LIN {X 0,Y 116.665,Z 500.549,A -85,B 0,C 180,E1 -26190.852,E2 -26190.852} C_VEL
LIN {X 0,Y 112.984,Z 509.27,A -85,B 0,C 180,E1 -26195.582,E2 -26195.582} C_VEL
LIN {X 0,Y 109.778,Z 516.952,A -85,B 0,C 180,E1 -26201.06,E2 -26201.06} C_VEL
LIN {X 0,Y 107.278,Z 523.285,A -85,B 0,C 180,E1 -26207.132,E2 -26207.132} C_VEL
LIN {X 0,Y 105.67,Z 528.207,A -85,B 0,C 180,E1 -26213.504,E2 -26213.504} C_VEL
LIN {X 0,Y 104.773,Z 531.45,A -85,B 0,C 180,E1 -26219.305,E2 -26219.305} C_VEL
LIN {X 0,Y 105.042,Z 534.238,A -85,B 0,C 180,E1 -26227.006,E2 -26227.006} C_VEL
LIN {X 0,Y 106.467,Z 535.327,A -85,B 0,C 180,E1 -26233.438,E2 -26233.438} C_VEL
LIN {X 0,Y 109.318,Z 535.217,A -85,B 0,C 180,E1 -26240.463,E2 -26240.463} C_VEL
LIN {X 0,Y 112.597,Z 534.109,A -85,B 0,C 180,E1 -26245.822,E2 -26245.822} C_VEL
LIN {X 0,Y 117.145,Z 531.835,A -85,B 0,C 180,E1 -26251.317,E2 -26251.317} C_VEL
LIN {X 0,Y 122.747,Z 528.36,A -85,B 0,C 180,E1 -26256.372,E2 -26256.372} C_VEL
LIN {X 0,Y 129.145,Z 523.621,A -85,B 0,C 180,E1 -26260.942,E2 -26260.942} C_VEL
LIN {X 0,Y 136.15,Z 517.469,A -85,B 0,C 180,E1 -26265.043,E2 -26265.043} C_VEL
LIN {X 0,Y 143.911,Z 509.526,A -85,B 0,C 180,E1 -26268.735,E2 -26268.735} C_VEL
LIN {X 0,Y 150.719,Z 501.38,A -85,B 0,C 180,E1 -26271.527,E2 -26271.527} C_VEL
LIN {X 0,Y 157.259,Z 492.279,A -85,B 0,C 180,E1 -26273.801,E2 -26273.801} C_VEL
LIN {X 0,Y 163.793,Z 481.328,A -85,B 0,C 180,E1 -26275.864,E2 -26275.864} C_VEL
LIN {X 0,Y 169.141,Z 470.396,A -85,B 0,C 180,E1 -26277.418,E2 -26277.418} C_VEL
LIN {X 0,Y 173.622,Z 458.97,A -85,B 0,C 180,E1 -26278.608,E2 -26278.608} C_VEL
LIN {X 0,Y 177.377,Z 446.045,A -85,B 0,C 180,E1 -26279.628,E2 -26279.628} C_VEL
LIN {X 0,Y 180.062,Z 433.099,A -85,B 0,C 180,E1 -26280.239,E2 -26280.239} C_VEL
LIN {X 0,Y 181.656,Z 420.065,A -85,B 0,C 180,E1 -26280.703,E2 -26280.703} C_VEL
LIN {X 0,Y 179.793,Z 415.381,A -85,B 0,C 180,E1 -26283.473,E2 -26283.473} C_VEL
LIN {X 0,Y 178.027,Z 411.229,A -85,B 0,C 180,E1 -26286.802,E2 -26286.802} C_VEL
LIN {X 0,Y 177.28,Z 409.415,A -85,B 0,C 180,E1 -26288.729,E2 -26288.729} C_VEL
LIN {X 0,Y 176.009,Z 407.916,A -85,B 0,C 180,E1 -26293.862,E2 -26293.862} C_VEL
LIN {X 0,Y 175.948,Z 407.96,A -85,B 0,C 180,E1 -26297.086,E2 -26297.086} C_VEL
LIN {X 0,Y 176.976,Z 409.546,A -85,B 0,C 180,E1 -26302.087,E2 -26302.087} C_VEL
LIN {X 0,Y 178.38,Z 414.032,A -85,B 0,C 180,E1 -26305.887,E2 -26305.887} C_VEL
LIN {X 0,Y 179.645,Z 417.893,A -85,B 0,C 180,E1 -26308.255,E2 -26308.255} C_VEL
LIN {X 0,Y 181.323,Z 423.803,A -85,B 0,C 180,E1 -26310.965,E2 -26310.965} C_VEL
LIN {X 0,Y 178.937,Z 441.292,A -85,B 0,C 180,E1 -26311.578,E2 -26311.578} C_VEL
LIN {X 0,Y 175.823,Z 454.417,A -85,B 0,C 180,E1 -26312.249,E2 -26312.249} C_VEL
LIN {X 0,Y 171.93,Z 466.104,A -85,B 0,C 180,E1 -26313.093,E2 -26313.093} C_VEL
LIN {X 0,Y 166.888,Z 477.934,A -85,B 0,C 180,E1 -26314.284,E2 -26314.284} C_VEL
LIN {X 0,Y 161.219,Z 488.681,A -85,B 0,C 180,E1 -26315.736,E2 -26315.736} C_VEL
LIN {X 0,Y 155.145,Z 498.423,A -85,B 0,C 180,E1 -26317.576,E2 -26317.576} C_VEL
LIN {X 0,Y 148.601,Z 507.346,A -85,B 0,C 180,E1 -26319.796,E2 -26319.796} C_VEL
LIN {X 0,Y 142.303,Z 514.803,A -85,B 0,C 180,E1 -26322.217,E2 -26322.217} C_VEL
LIN {X 0,Y 135.314,Z 522.176,A -85,B 0,C 180,E1 -26325.497,E2 -26325.497} C_VEL
LIN {X 0,Y 128.731,Z 528.172,A -85,B 0,C 180,E1 -26329.087,E2 -26329.087} C_VEL
LIN {X 0,Y 122.68,Z 533.16,A -85,B 0,C 180,E1 -26333.323,E2 -26333.323} C_VEL
LIN {X 0,Y 117.749,Z 536.703,A -85,B 0,C 180,E1 -26337.524,E2 -26337.524} C_VEL
LIN {X 0,Y 112.044,Z 540.244,A -85,B 0,C 180,E1 -26343.97,E2 -26343.97} C_VEL
LIN {X 0,Y 107.971,Z 542.164,A -85,B 0,C 180,E1 -26351.021,E2 -26351.021} C_VEL
LIN {X 0,Y 105.791,Z 542.603,A -85,B 0,C 180,E1 -26358.518,E2 -26358.518} C_VEL
LIN {X 0,Y 105.297,Z 542.259,A -85,B 0,C 180,E1 -26362.342,E2 -26362.342} C_VEL
LIN {X 0,Y 105.199,Z 541.5,A -85,B 0,C 180,E1 -26366.182,E2 -26366.182} C_VEL
LIN {X 0,Y 105.382,Z 540.344,A -85,B 0,C 180,E1 -26370.012,E2 -26370.012} C_VEL
LIN {X 0,Y 105.287,Z 537.737,A -85,B 0,C 180,E1 -26375.759,E2 -26375.759} C_VEL
LIN {X 0,Y 105.847,Z 534.06,A -85,B 0,C 180,E1 -26381.502,E2 -26381.502} C_VEL
LIN {X 0,Y 107.216,Z 529.214,A -85,B 0,C 180,E1 -26387.168,E2 -26387.168} C_VEL
LIN {X 0,Y 109.582,Z 523.072,A -85,B 0,C 180,E1 -26392.643,E2 -26392.643} C_VEL
LIN {X 0,Y 112.775,Z 515.39,A -85,B 0,C 180,E1 -26397.876,E2 -26397.876} C_VEL
LIN {X 0,Y 115.509,Z 508.774,A -85,B 0,C 180,E1 -26401.396,E2 -26401.396} C_VEL
LIN {X 0,Y 119.502,Z 498.92,A -85,B 0,C 180,E1 -26405.514,E2 -26405.514} C_VEL
LIN {X 0,Y 123.418,Z 488.458,A -85,B 0,C 180,E1 -26408.795,E2 -26408.795} C_VEL
LIN {X 0,Y 127.343,Z 476.934,A -85,B 0,C 180,E1 -26411.484,E2 -26411.484} C_VEL
LIN {X 0,Y 129.324,Z 469.742,A -85,B 0,C 180,E1 -26412.819,E2 -26412.819} C_VEL
LIN {X 0,Y 130.256,Z 464.373,A -85,B 0,C 180,E1 -26413.78,E2 -26413.78} C_VEL
LIN {X 0,Y 129.985,Z 455.35,A -85,B 0,C 180,E1 -26415.619,E2 -26415.619} C_VEL
LIN {X 0,Y 129.24,Z 446.167,A -85,B 0,C 180,E1 -26417.279,E2 -26417.279} C_VEL
LIN {X 0,Y 129.425,Z 440.424,A -85,B 0,C 180,E1 -26417.922,E2 -26417.922} C_VEL
LIN {X 0,Y 132.785,Z 401.785,A -85,B 0,C 180,E1 -26419.9,E2 -26419.9} C_VEL
LIN {X 0,Y 132.575,Z 398.319,A -85,B 0,C 180,E1 -26420.249,E2 -26420.249} C_VEL
LIN {X 0,Y 127.688,Z 383.599,A -85,B 0,C 180,E1 -26423.302,E2 -26423.302} C_VEL
LIN {X 0,Y 122.637,Z 371.093,A -85,B 0,C 180,E1 -26426.647,E2 -26426.647} C_VEL
LIN {X 0,Y 118.748,Z 363.954,A -85,B 0,C 180,E1 -26429.275,E2 -26429.275} C_VEL
LIN {X 0,Y 113.441,Z 355.782,A -85,B 0,C 180,E1 -26433.186,E2 -26433.186} C_VEL
LIN {X 0,Y 111.169,Z 352.453,A -85,B 0,C 180,E1 -26435.068,E2 -26435.068} C_VEL
LIN {X 0,Y 108.638,Z 348.864,A -85,B 0,C 180,E1 -26437.286,E2 -26437.286} C_VEL
LIN {X 0,Y 105.705,Z 345.199,A -85,B 0,C 180,E1 -26440.078,E2 -26440.078} C_VEL
LIN {X 0,Y 104.68,Z 343.35,A -85,B 0,C 180,E1 -26441.226,E2 -26441.226} C_VEL
LIN {X 0,Y 102.272,Z 341.321,A -85,B 0,C 180,E1 -26443.808,E2 -26443.808} C_VEL
LIN {X 0,Y 101.161,Z 338.839,A -85,B 0,C 180,E1 -26445.351,E2 -26445.351} C_VEL
LIN {X 0,Y 100.982,Z 337.862,A -85,B 0,C 180,E1 -26445.818,E2 -26445.818} C_VEL
LIN {X 0,Y 101.24,Z 337.863,A -85,B 0,C 180,E1 -26452.019,E2 -26452.019} C_VEL
LIN {X 0,Y 101.844,Z 337.735,A -85,B 0,C 180,E1 -26460,E2 -26460} C_VEL
LIN {X 0,Y 101.234,Z 337.865,A -85,B 0,C 180,E1 -26467.981,E2 -26467.981} C_VEL
LIN {X 0,Y 101.064,Z 337.89,A -85,B 0,C 180,E1 -26473.164,E2 -26473.164} C_VEL
LIN {X 0,Y 100.778,Z 337.914,A -85,B 0,C 180,E1 -26480.407,E2 -26480.407} C_VEL
LIN {X 0,Y 100.715,Z 337.93,A -85,B 0,C 180,E1 -26484.863,E2 -26484.863} C_VEL
LIN {X 0,Y 100.651,Z 337.879,A -85,B 0,C 180,E1 -26493.063,E2 -26493.063} C_VEL
LIN {X 0,Y 100.637,Z 337.948,A -85,B 0,C 180,E1 -26499.793,E2 -26499.793} C_VEL
LIN {X 0,Y 100.608,Z 337.953,A -85,B 0,C 180,E1 -26506.537,E2 -26506.537} C_VEL
LIN {X 0,Y 101.477,Z 340.593,A -85,B 0,C 180,E1 -26507.943,E2 -26507.943} C_VEL
LIN {X 0,Y 103.656,Z 342.892,A -85,B 0,C 180,E1 -26510.43,E2 -26510.43} C_VEL
LIN {X 0,Y 104.88,Z 343.867,A -85,B 0,C 180,E1 -26511.687,E2 -26511.687} C_VEL
LIN {X 0,Y 106.673,Z 346.893,A -85,B 0,C 180,E1 -26513.621,E2 -26513.621} C_VEL
LIN {X 0,Y 108.718,Z 349.01,A -85,B 0,C 180,E1 -26515.473,E2 -26515.473} C_VEL
LIN {X 0,Y 111.229,Z 352.53,A -85,B 0,C 180,E1 -26517.66,E2 -26517.66} C_VEL
LIN {X 0,Y 115.759,Z 359.291,A -85,B 0,C 180,E1 -26521.274,E2 -26521.274} C_VEL
LIN {X 0,Y 119.958,Z 365.783,A -85,B 0,C 180,E1 -26524.211,E2 -26524.211} C_VEL
LIN {X 0,Y 126.98,Z 378.193,A -85,B 0,C 180,E1 -26528.608,E2 -26528.608} C_VEL
LIN {X 0,Y 133.38,Z 392.007,A -85,B 0,C 180,E1 -26532.218,E2 -26532.218} C_VEL
LIN {X 0,Y 129.761,Z 432.259,A -85,B 0,C 180,E1 -26534.216,E2 -26534.216} C_VEL
LIN {X 0,Y 127.732,Z 445.85,A -85,B 0,C 180,E1 -26535.452,E2 -26535.452} C_VEL
LIN {X 0,Y 124.976,Z 458.682,A -85,B 0,C 180,E1 -26537.197,E2 -26537.197} C_VEL
LIN {X 0,Y 121.513,Z 470.852,A -85,B 0,C 180,E1 -26539.497,E2 -26539.497} C_VEL
LIN {X 0,Y 117.767,Z 481.821,A -85,B 0,C 180,E1 -26542.273,E2 -26542.273} C_VEL
LIN {X 0,Y 113.927,Z 491.71,A -85,B 0,C 180,E1 -26545.566,E2 -26545.566} C_VEL
LIN {X 0,Y 109.663,Z 501.7,A -85,B 0,C 180,E1 -26549.988,E2 -26549.988} C_VEL
LIN {X 0,Y 105.832,Z 510.342,A -85,B 0,C 180,E1 -26555.052,E2 -26555.052} C_VEL
LIN {X 0,Y 102.535,Z 517.772,A -85,B 0,C 180,E1 -26560.851,E2 -26560.851} C_VEL
LIN {X 0,Y 100.35,Z 523.077,A -85,B 0,C 180,E1 -26566.254,E2 -26566.254} C_VEL
LIN {X 0,Y 98.774,Z 527.651,A -85,B 0,C 180,E1 -26572.333,E2 -26572.333} C_VEL
LIN {X 0,Y 97.814,Z 530.795,A -85,B 0,C 180,E1 -26577.824,E2 -26577.824} C_VEL
LIN {X 0,Y 97.714,Z 533.677,A -85,B 0,C 180,E1 -26585.108,E2 -26585.108} C_VEL
LIN {X 0,Y 98.401,Z 534.905,A -85,B 0,C 180,E1 -26589.98,E2 -26589.98} C_VEL
LIN {X 0,Y 99.836,Z 535.622,A -85,B 0,C 180,E1 -26595.254,E2 -26595.254} C_VEL
LIN {X 0,Y 102.768,Z 535.548,A -85,B 0,C 180,E1 -26602.013,E2 -26602.013} C_VEL
LIN {X 0,Y 107.044,Z 534.256,A -85,B 0,C 180,E1 -26608.566,E2 -26608.566} C_VEL
LIN {X 0,Y 111.831,Z 532.052,A -85,B 0,C 180,E1 -26613.902,E2 -26613.902} C_VEL
LIN {X 0,Y 117.929,Z 528.545,A -85,B 0,C 180,E1 -26619.049,E2 -26619.049} C_VEL
LIN {X 0,Y 124.838,Z 523.752,A -85,B 0,C 180,E1 -26623.651,E2 -26623.651} C_VEL
LIN {X 0,Y 132.368,Z 517.529,A -85,B 0,C 180,E1 -26627.738,E2 -26627.738} C_VEL
LIN {X 0,Y 140.548,Z 509.577,A -85,B 0,C 180,E1 -26631.372,E2 -26631.372} C_VEL
LIN {X 0,Y 148.293,Z 500.616,A -85,B 0,C 180,E1 -26634.283,E2 -26634.283} C_VEL
LIN {X 0,Y 154.89,Z 491.628,A -85,B 0,C 180,E1 -26636.388,E2 -26636.388} C_VEL
LIN {X 0,Y 161.675,Z 480.485,A -85,B 0,C 180,E1 -26638.372,E2 -26638.372} C_VEL
LIN {X 0,Y 167.387,Z 468.939,A -85,B 0,C 180,E1 -26639.869,E2 -26639.869} C_VEL
LIN {X 0,Y 172.181,Z 456.516,A -85,B 0,C 180,E1 -26641.067,E2 -26641.067} C_VEL
LIN {X 0,Y 175.631,Z 444.538,A -85,B 0,C 180,E1 -26641.915,E2 -26641.915} C_VEL
LIN {X 0,Y 178.261,Z 431.148,A -85,B 0,C 180,E1 -26642.472,E2 -26642.472} C_VEL
LIN {X 0,Y 179.109,Z 424.236,A -85,B 0,C 180,E1 -26642.752,E2 -26642.752} C_VEL
LIN {X 0,Y 177.663,Z 420.643,A -85,B 0,C 180,E1 -26645.224,E2 -26645.224} C_VEL
LIN {X 0,Y 176.617,Z 417.72,A -85,B 0,C 180,E1 -26647.664,E2 -26647.664} C_VEL
LIN {X 0,Y 176.084,Z 416.319,A -85,B 0,C 180,E1 -26649.187,E2 -26649.187} C_VEL
LIN {X 0,Y 175.003,Z 414.923,A -85,B 0,C 180,E1 -26653.943,E2 -26653.943} C_VEL
LIN {X 0,Y 174.957,Z 415.009,A -85,B 0,C 180,E1 -26657.186,E2 -26657.186} C_VEL
LIN {X 0,Y 175.803,Z 416.417,A -85,B 0,C 180,E1 -26661.627,E2 -26661.627} C_VEL
LIN {X 0,Y 177.023,Z 420.909,A -85,B 0,C 180,E1 -26665.342,E2 -26665.342} C_VEL
LIN {X 0,Y 178.184,Z 424.879,A -85,B 0,C 180,E1 -26667.725,E2 -26667.725} C_VEL
LIN {X 0,Y 178.797,Z 427.471,A -85,B 0,C 180,E1 -26668.905,E2 -26668.905} C_VEL
LIN {X 0,Y 176.708,Z 441.516,A -85,B 0,C 180,E1 -26669.408,E2 -26669.408} C_VEL
LIN {X 0,Y 173.682,Z 453.811,A -85,B 0,C 180,E1 -26670.006,E2 -26670.006} C_VEL
LIN {X 0,Y 169.713,Z 465.425,A -85,B 0,C 180,E1 -26670.786,E2 -26670.786} C_VEL
LIN {X 0,Y 164.502,Z 477.304,A -85,B 0,C 180,E1 -26671.906,E2 -26671.906} C_VEL
LIN {X 0,Y 157.966,Z 489.289,A -85,B 0,C 180,E1 -26673.488,E2 -26673.488} C_VEL
LIN {X 0,Y 150.979,Z 499.835,A -85,B 0,C 180,E1 -26675.471,E2 -26675.471} C_VEL
LIN {X 0,Y 144.214,Z 508.486,A -85,B 0,C 180,E1 -26677.656,E2 -26677.656} C_VEL
LIN {X 0,Y 137.676,Z 515.698,A -85,B 0,C 180,E1 -26680.049,E2 -26680.049} C_VEL
LIN {X 0,Y 130.37,Z 522.837,A -85,B 0,C 180,E1 -26683.32,E2 -26683.32} C_VEL
LIN {X 0,Y 123.463,Z 528.639,A -85,B 0,C 180,E1 -26686.933,E2 -26686.933} C_VEL
LIN {X 0,Y 116.658,Z 533.752,A -85,B 0,C 180,E1 -26691.552,E2 -26691.552} C_VEL
LIN {X 0,Y 111.833,Z 536.868,A -85,B 0,C 180,E1 -26695.574,E2 -26695.574} C_VEL
LIN {X 0,Y 108.521,Z 538.758,A -85,B 0,C 180,E1 -26698.812,E2 -26698.812} C_VEL
LIN {X 0,Y 103.228,Z 541.282,A -85,B 0,C 180,E1 -26705.905,E2 -26705.905} C_VEL
LIN {X 0,Y 99.829,Z 542.33,A -85,B 0,C 180,E1 -26713.659,E2 -26713.659} C_VEL
LIN {X 0,Y 98.838,Z 542.292,A -85,B 0,C 180,E1 -26717.698,E2 -26717.698} C_VEL
LIN {X 0,Y 98.111,Z 541.02,A -85,B 0,C 180,E1 -26725.906,E2 -26725.906} C_VEL
LIN {X 0,Y 98.305,Z 539.804,A -85,B 0,C 180,E1 -26730.013,E2 -26730.013} C_VEL
LIN {X 0,Y 98.221,Z 537.073,A -85,B 0,C 180,E1 -26736.174,E2 -26736.174} C_VEL
LIN {X 0,Y 98.884,Z 533.268,A -85,B 0,C 180,E1 -26742.324,E2 -26742.324} C_VEL
LIN {X 0,Y 100.421,Z 528.285,A -85,B 0,C 180,E1 -26748.369,E2 -26748.369} C_VEL
LIN {X 0,Y 103.044,Z 521.999,A -85,B 0,C 180,E1 -26754.168,E2 -26754.168} C_VEL
LIN {X 0,Y 106.495,Z 514.07,A -85,B 0,C 180,E1 -26759.678,E2 -26759.678} C_VEL
LIN {X 0,Y 110.42,Z 505.227,A -85,B 0,C 180,E1 -26764.308,E2 -26764.308} C_VEL
LIN {X 0,Y 114.237,Z 496.074,A -85,B 0,C 180,E1 -26767.979,E2 -26767.979} C_VEL
LIN {X 0,Y 118.457,Z 485.04,A -85,B 0,C 180,E1 -26771.314,E2 -26771.314} C_VEL
LIN {X 0,Y 122.03,Z 474.28,A -85,B 0,C 180,E1 -26773.729,E2 -26773.729} C_VEL
LIN {X 0,Y 125.551,Z 461.419,A -85,B 0,C 180,E1 -26775.836,E2 -26775.836} C_VEL
LIN {X 0,Y 128.155,Z 448.849,A -85,B 0,C 180,E1 -26777.257,E2 -26777.257} C_VEL
LIN {X 0,Y 129.425,Z 440.424,A -85,B 0,C 180,E1 -26777.922,E2 -26777.922} C_VEL
LIN {X 0,Y 129.569,Z 434.661,A -85,B 0,C 180,E1 -26778.478,E2 -26778.478} C_VEL
LIN {X 0,Y 126.8,Z 415.841,A -85,B 0,C 180,E1 -26780.976,E2 -26780.976} C_VEL
LIN {X 0,Y 126.704,Z 410.024,A -85,B 0,C 180,E1 -26781.472,E2 -26781.472} C_VEL
LIN {X 0,Y 127.263,Z 400.819,A -85,B 0,C 180,E1 -26782.022,E2 -26782.022} C_VEL
LIN {X 0,Y 122.632,Z 386.514,A -85,B 0,C 180,E1 -26785.221,E2 -26785.221} C_VEL
LIN {X 0,Y 117.719,Z 374.148,A -85,B 0,C 180,E1 -26788.789,E2 -26788.789} C_VEL
LIN {X 0,Y 112.832,Z 365.521,A -85,B 0,C 180,E1 -26792.465,E2 -26792.465} C_VEL
LIN {X 0,Y 108.275,Z 358.439,A -85,B 0,C 180,E1 -26796.346,E2 -26796.346} C_VEL
LIN {X 0,Y 104.809,Z 353.675,A -85,B 0,C 180,E1 -26799.643,E2 -26799.643} C_VEL
LIN {X 0,Y 102.41,Z 350.065,A -85,B 0,C 180,E1 -26802.299,E2 -26802.299} C_VEL
LIN {X 0,Y 99.45,Z 346.857,A -85,B 0,C 180,E1 -26805.81,E2 -26805.81} C_VEL
LIN {X 0,Y 98.251,Z 344.352,A -85,B 0,C 180,E1 -26807.608,E2 -26807.608} C_VEL
LIN {X 0,Y 95.865,Z 342.587,A -85,B 0,C 180,E1 -26811.038,E2 -26811.038} C_VEL
LIN {X 0,Y 94.427,Z 339.863,A -85,B 0,C 180,E1 -26813.858,E2 -26813.858} C_VEL
LIN {X 0,Y 94.233,Z 338.69,A -85,B 0,C 180,E1 -26814.651,E2 -26814.651} C_VEL
LIN {X 0,Y 94.773,Z 338.613,A -85,B 0,C 180,E1 -26820,E2 -26820} C_VEL
LIN {X 0,Y 94.145,Z 338.742,A -85,B 0,C 180,E1 -26828.587,E2 -26828.587} C_VEL
LIN {X 0,Y 93.972,Z 338.775,A -85,B 0,C 180,E1 -26833.487,E2 -26833.487} C_VEL
LIN {X 0,Y 93.645,Z 338.814,A -85,B 0,C 180,E1 -26842.04,E2 -26842.04} C_VEL
LIN {X 0,Y 93.555,Z 338.791,A -85,B 0,C 180,E1 -26846.791,E2 -26846.791} C_VEL
LIN {X 0,Y 93.556,Z 338.77,A -85,B 0,C 180,E1 -26854.257,E2 -26854.257} C_VEL
LIN {X 0,Y 93.533,Z 338.972,A -85,B 0,C 180,E1 -26857.071,E2 -26857.071} C_VEL
LIN {X 0,Y 94.242,Z 341.088,A -85,B 0,C 180,E1 -26858.806,E2 -26858.806} C_VEL
LIN {X 0,Y 96.082,Z 343.431,A -85,B 0,C 180,E1 -26862.095,E2 -26862.095} C_VEL
LIN {X 0,Y 98.178,Z 344.839,A -85,B 0,C 180,E1 -26865.067,E2 -26865.067} C_VEL
LIN {X 0,Y 99.749,Z 347.721,A -85,B 0,C 180,E1 -26867.341,E2 -26867.341} C_VEL
LIN {X 0,Y 102.304,Z 350.218,A -85,B 0,C 180,E1 -26870.284,E2 -26870.284} C_VEL
LIN {X 0,Y 104.479,Z 353.509,A -85,B 0,C 180,E1 -26872.729,E2 -26872.729} C_VEL
LIN {X 0,Y 106.069,Z 355.432,A -85,B 0,C 180,E1 -26874.296,E2 -26874.296} C_VEL
LIN {X 0,Y 109.432,Z 360.383,A -85,B 0,C 180,E1 -26877.391,E2 -26877.391} C_VEL
LIN {X 0,Y 113.983,Z 367.303,A -85,B 0,C 180,E1 -26881.098,E2 -26881.098} C_VEL
LIN {X 0,Y 120.248,Z 378.29,A -85,B 0,C 180,E1 -26885.559,E2 -26885.559} C_VEL
LIN {X 0,Y 124.203,Z 386.015,A -85,B 0,C 180,E1 -26888.1,E2 -26888.1} C_VEL
LIN {X 0,Y 127.722,Z 394.162,A -85,B 0,C 180,E1 -26890.271,E2 -26890.271} C_VEL
LIN {X 0,Y 124.17,Z 432.589,A -85,B 0,C 180,E1 -26892.243,E2 -26892.243} C_VEL
LIN {X 0,Y 122.087,Z 445.935,A -85,B 0,C 180,E1 -26893.477,E2 -26893.477} C_VEL
LIN {X 0,Y 119.216,Z 458.812,A -85,B 0,C 180,E1 -26895.262,E2 -26895.262} C_VEL
LIN {X 0,Y 115.342,Z 471.772,A -85,B 0,C 180,E1 -26897.791,E2 -26897.791} C_VEL
LIN {X 0,Y 111.105,Z 483.373,A -85,B 0,C 180,E1 -26900.89,E2 -26900.89} C_VEL
LIN {X 0,Y 106.412,Z 494.631,A -85,B 0,C 180,E1 -26905.03,E2 -26905.03} C_VEL
LIN {X 0,Y 101.85,Z 504.567,A -85,B 0,C 180,E1 -26909.987,E2 -26909.987} C_VEL
LIN {X 0,Y 98.237,Z 512.27,A -85,B 0,C 180,E1 -26915.14,E2 -26915.14} C_VEL
LIN {X 0,Y 94.783,Z 519.726,A -85,B 0,C 180,E1 -26921.751,E2 -26921.751} C_VEL
LIN {X 0,Y 92.75,Z 524.709,A -85,B 0,C 180,E1 -26927.628,E2 -26927.628} C_VEL
LIN {X 0,Y 91.123,Z 529.462,A -85,B 0,C 180,E1 -26935.08,E2 -26935.08} C_VEL
LIN {X 0,Y 90.508,Z 532.89,A -85,B 0,C 180,E1 -26942.906,E2 -26942.906} C_VEL
LIN {X 0,Y 91.201,Z 534.814,A -85,B 0,C 180,E1 -26949.592,E2 -26949.592} C_VEL
LIN {X 0,Y 93.339,Z 535.914,A -85,B 0,C 180,E1 -26957.339,E2 -26957.339} C_VEL
LIN {X 0,Y 96.695,Z 535.815,A -85,B 0,C 180,E1 -26964.447,E2 -26964.447} C_VEL
LIN {X 0,Y 101.187,Z 534.601,A -85,B 0,C 180,E1 -26970.909,E2 -26970.909} C_VEL
LIN {X 0,Y 106.958,Z 532.196,A -85,B 0,C 180,E1 -26976.872,E2 -26976.872} C_VEL
LIN {X 0,Y 113.405,Z 528.751,A -85,B 0,C 180,E1 -26981.949,E2 -26981.949} C_VEL
LIN {X 0,Y 120.858,Z 523.923,A -85,B 0,C 180,E1 -26986.549,E2 -26986.549} C_VEL
LIN {X 0,Y 128.934,Z 517.602,A -85,B 0,C 180,E1 -26990.588,E2 -26990.588} C_VEL
LIN {X 0,Y 137.509,Z 509.619,A -85,B 0,C 180,E1 -26994.133,E2 -26994.133} C_VEL
LIN {X 0,Y 145.148,Z 501.198,A -85,B 0,C 180,E1 -26996.768,E2 -26996.768} C_VEL
LIN {X 0,Y 152.847,Z 491.087,A -85,B 0,C 180,E1 -26999.034,E2 -26999.034} C_VEL
LIN {X 0,Y 159.337,Z 480.758,A -85,B 0,C 180,E1 -27000.789,E2 -27000.789} C_VEL
LIN {X 0,Y 165.215,Z 469.244,A -85,B 0,C 180,E1 -27002.211,E2 -27002.211} C_VEL
LIN {X 0,Y 170.202,Z 456.677,A -85,B 0,C 180,E1 -27003.368,E2 -27003.368} C_VEL
LIN {X 0,Y 173.868,Z 444.229,A -85,B 0,C 180,E1 -27004.187,E2 -27004.187} C_VEL
LIN {X 0,Y 176.467,Z 431.106,A -85,B 0,C 180,E1 -27004.685,E2 -27004.685} C_VEL
LIN {X 0,Y 176.792,Z 428.711,A -85,B 0,C 180,E1 -27004.793,E2 -27004.793} C_VEL
LIN {X 0,Y 175.338,Z 424.442,A -85,B 0,C 180,E1 -27008.282,E2 -27008.282} C_VEL
LIN {X 0,Y 174.758,Z 423.035,A -85,B 0,C 180,E1 -27010.067,E2 -27010.067} C_VEL
LIN {X 0,Y 173.975,Z 421.931,A -85,B 0,C 180,E1 -27014.229,E2 -27014.229} C_VEL
LIN {X 0,Y 173.963,Z 422.087,A -85,B 0,C 180,E1 -27017.287,E2 -27017.287} C_VEL
LIN {X 0,Y 174.653,Z 423.395,A -85,B 0,C 180,E1 -27021.233,E2 -27021.233} C_VEL
LIN {X 0,Y 175.67,Z 427.597,A -85,B 0,C 180,E1 -27024.681,E2 -27024.681} C_VEL
LIN {X 0,Y 176.53,Z 431.263,A -85,B 0,C 180,E1 -27026.802,E2 -27026.802} C_VEL
LIN {X 0,Y 174.269,Z 443.994,A -85,B 0,C 180,E1 -27027.26,E2 -27027.26} C_VEL
LIN {X 0,Y 170.647,Z 457.145,A -85,B 0,C 180,E1 -27027.93,E2 -27027.93} C_VEL
LIN {X 0,Y 166.284,Z 468.708,A -85,B 0,C 180,E1 -27028.741,E2 -27028.741} C_VEL
LIN {X 0,Y 160.965,Z 479.778,A -85,B 0,C 180,E1 -27029.822,E2 -27029.822} C_VEL
LIN {X 0,Y 154.23,Z 491.13,A -85,B 0,C 180,E1 -27031.329,E2 -27031.329} C_VEL
LIN {X 0,Y 147.028,Z 501.279,A -85,B 0,C 180,E1 -27033.249,E2 -27033.249} C_VEL
LIN {X 0,Y 138.691,Z 511.07,A -85,B 0,C 180,E1 -27035.85,E2 -27035.85} C_VEL
LIN {X 0,Y 133.26,Z 516.604,A -85,B 0,C 180,E1 -27037.734,E2 -27037.734} C_VEL
LIN {X 0,Y 125.632,Z 523.503,A -85,B 0,C 180,E1 -27040.977,E2 -27040.977} C_VEL
LIN {X 0,Y 118.392,Z 529.106,A -85,B 0,C 180,E1 -27044.594,E2 -27044.594} C_VEL
LIN {X 0,Y 110.781,Z 534.254,A -85,B 0,C 180,E1 -27049.578,E2 -27049.578} C_VEL
LIN {X 0,Y 106.043,Z 537.026,A -85,B 0,C 180,E1 -27053.4,E2 -27053.4} C_VEL
LIN {X 0,Y 102.504,Z 538.794,A -85,B 0,C 180,E1 -27056.753,E2 -27056.753} C_VEL
LIN {X 0,Y 96.784,Z 541.179,A -85,B 0,C 180,E1 -27064.188,E2 -27064.188} C_VEL
LIN {X 0,Y 94.585,Z 541.817,A -85,B 0,C 180,E1 -27068.207,E2 -27068.207} C_VEL
LIN {X 0,Y 91.882,Z 541.932,A -85,B 0,C 180,E1 -27076.75,E2 -27076.75} C_VEL
LIN {X 0,Y 91.04,Z 540.541,A -85,B 0,C 180,E1 -27085.587,E2 -27085.587} C_VEL
LIN {X 0,Y 91.215,Z 539.262,A -85,B 0,C 180,E1 -27090.014,E2 -27090.014} C_VEL
LIN {X 0,Y 91.178,Z 536.404,A -85,B 0,C 180,E1 -27096.653,E2 -27096.653} C_VEL
LIN {X 0,Y 91.953,Z 532.461,A -85,B 0,C 180,E1 -27103.269,E2 -27103.269} C_VEL
LIN {X 0,Y 94.061,Z 526.314,A -85,B 0,C 180,E1 -27110.801,E2 -27110.801} C_VEL
LIN {X 0,Y 97.096,Z 519.568,A -85,B 0,C 180,E1 -27116.91,E2 -27116.91} C_VEL
LIN {X 0,Y 101.007,Z 511.143,A -85,B 0,C 180,E1 -27122.645,E2 -27122.645} C_VEL
LIN {X 0,Y 105.05,Z 502.467,A -85,B 0,C 180,E1 -27127.034,E2 -27127.034} C_VEL
LIN {X 0,Y 109.683,Z 491.788,A -85,B 0,C 180,E1 -27131.067,E2 -27131.067} C_VEL
LIN {X 0,Y 113.774,Z 481.222,A -85,B 0,C 180,E1 -27134.034,E2 -27134.034} C_VEL
LIN {X 0,Y 117.534,Z 469.483,A -85,B 0,C 180,E1 -27136.482,E2 -27136.482} C_VEL
LIN {X 0,Y 121.012,Z 456.231,A -85,B 0,C 180,E1 -27138.407,E2 -27138.407} C_VEL
LIN {X 0,Y 123.437,Z 442.968,A -85,B 0,C 180,E1 -27139.716,E2 -27139.716} C_VEL
LIN {X 0,Y 124.987,Z 428.585,A -85,B 0,C 180,E1 -27140.583,E2 -27140.583} C_VEL
LIN {X 0,Y 126.704,Z 410.024,A -85,B 0,C 180,E1 -27141.472,E2 -27141.472} C_VEL
LIN {X 0,Y 126.409,Z 406.934,A -85,B 0,C 180,E1 -27141.844,E2 -27141.844} C_VEL
LIN {X 0,Y 124.852,Z 403.138,A -85,B 0,C 180,E1 -27142.79,E2 -27142.79} C_VEL
LIN {X 0,Y 119.609,Z 394.847,A -85,B 0,C 180,E1 -27145.852,E2 -27145.852} C_VEL
LIN {X 0,Y 118.966,Z 393.121,A -85,B 0,C 180,E1 -27146.326,E2 -27146.326} C_VEL
LIN {X 0,Y 114.902,Z 381.895,A -85,B 0,C 180,E1 -27149.496,E2 -27149.496} C_VEL
LIN {X 0,Y 112.445,Z 376.399,A -85,B 0,C 180,E1 -27151.486,E2 -27151.486} C_VEL
LIN {X 0,Y 107.195,Z 367.318,A -85,B 0,C 180,E1 -27156,E2 -27156} C_VEL
LIN {X 0,Y 104.558,Z 363.42,A -85,B 0,C 180,E1 -27158.499,E2 -27158.499} C_VEL
LIN {X 0,Y 101.95,Z 359.506,A -85,B 0,C 180,E1 -27161.288,E2 -27161.288} C_VEL
LIN {X 0,Y 99.407,Z 355.75,A -85,B 0,C 180,E1 -27164.363,E2 -27164.363} C_VEL
LIN {X 0,Y 97,Z 352.843,A -85,B 0,C 180,E1 -27167.517,E2 -27167.517} C_VEL
LIN {X 0,Y 95.944,Z 350.818,A -85,B 0,C 180,E1 -27169.221,E2 -27169.221} C_VEL
LIN {X 0,Y 93.656,Z 348.585,A -85,B 0,C 180,E1 -27172.996,E2 -27172.996} C_VEL
LIN {X 0,Y 92.25,Z 345.466,A -85,B 0,C 180,E1 -27176.178,E2 -27176.178} C_VEL
LIN {X 0,Y 89.759,Z 343.985,A -85,B 0,C 180,E1 -27182.244,E2 -27182.244} C_VEL
LIN {X 0,Y 87.815,Z 342.206,A -85,B 0,C 180,E1 -27191.542,E2 -27191.542} C_VEL
LIN {X 0,Y 87.56,Z 342.303,A -85,B 0,C 180,E1 -27197.519,E2 -27197.519} C_VEL
LIN {X 0,Y 88.537,Z 343.801,A -85,B 0,C 180,E1 -27206.273,E2 -27206.273} C_VEL
LIN {X 0,Y 91.71,Z 345.783,A -85,B 0,C 180,E1 -27215.572,E2 -27215.572} C_VEL
LIN {X 0,Y 93.334,Z 349.009,A -85,B 0,C 180,E1 -27219.256,E2 -27219.256} C_VEL
LIN {X 0,Y 96.005,Z 351.432,A -85,B 0,C 180,E1 -27223.653,E2 -27223.653} C_VEL
LIN {X 0,Y 98.151,Z 354.799,A -85,B 0,C 180,E1 -27226.842,E2 -27226.842} C_VEL
LIN {X 0,Y 99.878,Z 356.67,A -85,B 0,C 180,E1 -27228.959,E2 -27228.959} C_VEL
LIN {X 0,Y 102.316,Z 360.108,A -85,B 0,C 180,E1 -27231.802,E2 -27231.802} C_VEL
LIN {X 0,Y 106.016,Z 365.626,A -85,B 0,C 180,E1 -27235.605,E2 -27235.605} C_VEL
LIN {X 0,Y 110.606,Z 372.915,A -85,B 0,C 180,E1 -27239.647,E2 -27239.647} C_VEL
LIN {X 0,Y 116.454,Z 383.683,A -85,B 0,C 180,E1 -27244.187,E2 -27244.187} C_VEL
LIN {X 0,Y 120.174,Z 391.293,A -85,B 0,C 180,E1 -27246.748,E2 -27246.748} C_VEL
LIN {X 0,Y 122.315,Z 396.762,A -85,B 0,C 180,E1 -27248.232,E2 -27248.232} C_VEL
LIN {X 0,Y 118.78,Z 432.764,A -85,B 0,C 180,E1 -27250.083,E2 -27250.083} C_VEL
LIN {X 0,Y 116.533,Z 446.408,A -85,B 0,C 180,E1 -27251.361,E2 -27251.361} C_VEL
LIN {X 0,Y 113.599,Z 458.946,A -85,B 0,C 180,E1 -27253.131,E2 -27253.131} C_VEL
LIN {X 0,Y 109.652,Z 471.598,A -85,B 0,C 180,E1 -27255.639,E2 -27255.639} C_VEL
LIN {X 0,Y 105.081,Z 483.561,A -85,B 0,C 180,E1 -27258.902,E2 -27258.902} C_VEL
LIN {X 0,Y 100.583,Z 493.822,A -85,B 0,C 180,E1 -27262.754,E2 -27262.754} C_VEL
LIN {X 0,Y 95.745,Z 503.922,A -85,B 0,C 180,E1 -27267.883,E2 -27267.883} C_VEL
LIN {X 0,Y 91.555,Z 512.273,A -85,B 0,C 180,E1 -27273.694,E2 -27273.694} C_VEL
LIN {X 0,Y 88.109,Z 519.258,A -85,B 0,C 180,E1 -27280.212,E2 -27280.212} C_VEL
LIN {X 0,Y 85.818,Z 524.466,A -85,B 0,C 180,E1 -27286.639,E2 -27286.639} C_VEL
LIN {X 0,Y 84.045,Z 529.341,A -85,B 0,C 180,E1 -27294.696,E2 -27294.696} C_VEL
LIN {X 0,Y 83.416,Z 532.717,A -85,B 0,C 180,E1 -27302.592,E2 -27302.592} C_VEL
LIN {X 0,Y 84.472,Z 535.184,A -85,B 0,C 180,E1 -27311.704,E2 -27311.704} C_VEL
LIN {X 0,Y 86.969,Z 536.207,A -85,B 0,C 180,E1 -27319.723,E2 -27319.723} C_VEL
LIN {X 0,Y 91.247,Z 536.02,A -85,B 0,C 180,E1 -27327.879,E2 -27327.879} C_VEL
LIN {X 0,Y 95.877,Z 534.854,A -85,B 0,C 180,E1 -27333.908,E2 -27333.908} C_VEL
LIN {X 0,Y 102.089,Z 532.498,A -85,B 0,C 180,E1 -27339.866,E2 -27339.866} C_VEL
LIN {X 0,Y 109.246,Z 528.957,A -85,B 0,C 180,E1 -27345.088,E2 -27345.088} C_VEL
LIN {X 0,Y 117.208,Z 524.089,A -85,B 0,C 180,E1 -27349.637,E2 -27349.637} C_VEL
LIN {X 0,Y 125.819,Z 517.714,A -85,B 0,C 180,E1 -27353.586,E2 -27353.586} C_VEL
LIN {X 0,Y 134.887,Z 509.682,A -85,B 0,C 180,E1 -27357.013,E2 -27357.013} C_VEL
LIN {X 0,Y 143.164,Z 500.83,A -85,B 0,C 180,E1 -27359.623,E2 -27359.623} C_VEL
LIN {X 0,Y 151.138,Z 490.617,A -85,B 0,C 180,E1 -27361.738,E2 -27361.738} C_VEL
LIN {X 0,Y 157.479,Z 480.741,A -85,B 0,C 180,E1 -27363.301,E2 -27363.301} C_VEL
LIN {X 0,Y 163.758,Z 468.629,A -85,B 0,C 180,E1 -27364.701,E2 -27364.701} C_VEL
LIN {X 0,Y 168.983,Z 455.651,A -85,B 0,C 180,E1 -27365.802,E2 -27365.802} C_VEL
LIN {X 0,Y 172.463,Z 443.822,A -85,B 0,C 180,E1 -27366.507,E2 -27366.507} C_VEL
LIN {X 0,Y 174.623,Z 433.497,A -85,B 0,C 180,E1 -27366.935,E2 -27366.935} C_VEL
LIN {X 0,Y 174.034,Z 431.179,A -85,B 0,C 180,E1 -27368.879,E2 -27368.879} C_VEL
LIN {X 0,Y 173.616,Z 429.961,A -85,B 0,C 180,E1 -27370.406,E2 -27370.406} C_VEL
LIN {X 0,Y 172.991,Z 428.952,A -85,B 0,C 180,E1 -27374.108,E2 -27374.108} C_VEL
LIN {X 0,Y 173.008,Z 429.226,A -85,B 0,C 180,E1 -27377.779,E2 -27377.779} C_VEL
LIN {X 0,Y 173.454,Z 430.197,A -85,B 0,C 180,E1 -27380.599,E2 -27380.599} C_VEL
LIN {X 0,Y 174.238,Z 434.193,A -85,B 0,C 180,E1 -27383.946,E2 -27383.946} C_VEL
LIN {X 0,Y 174.407,Z 435.684,A -85,B 0,C 180,E1 -27384.714,E2 -27384.714} C_VEL
LIN {X 0,Y 171.458,Z 448.876,A -85,B 0,C 180,E1 -27385.184,E2 -27385.184} C_VEL
LIN {X 0,Y 167.023,Z 462.397,A -85,B 0,C 180,E1 -27385.914,E2 -27385.914} C_VEL
LIN {X 0,Y 161.478,Z 474.901,A -85,B 0,C 180,E1 -27386.872,E2 -27386.872} C_VEL
LIN {X 0,Y 154.522,Z 487.26,A -85,B 0,C 180,E1 -27388.236,E2 -27388.236} C_VEL
LIN {X 0,Y 147.74,Z 497.119,A -85,B 0,C 180,E1 -27389.78,E2 -27389.78} C_VEL
LIN {X 0,Y 140.406,Z 506.087,A -85,B 0,C 180,E1 -27391.711,E2 -27391.711} C_VEL
LIN {X 0,Y 131.827,Z 514.909,A -85,B 0,C 180,E1 -27394.299,E2 -27394.299} C_VEL
LIN {X 0,Y 123.763,Z 522.052,A -85,B 0,C 180,E1 -27397.367,E2 -27397.367} C_VEL
LIN {X 0,Y 116.004,Z 527.885,A -85,B 0,C 180,E1 -27400.795,E2 -27400.795} C_VEL
LIN {X 0,Y 108.866,Z 532.543,A -85,B 0,C 180,E1 -27404.776,E2 -27404.776} C_VEL
LIN {X 0,Y 103.296,Z 535.699,A -85,B 0,C 180,E1 -27408.655,E2 -27408.655} C_VEL
LIN {X 0,Y 96.637,Z 538.838,A -85,B 0,C 180,E1 -27414.442,E2 -27414.442} C_VEL
LIN {X 0,Y 90.416,Z 541.074,A -85,B 0,C 180,E1 -27422.219,E2 -27422.219} C_VEL
LIN {X 0,Y 86.232,Z 541.769,A -85,B 0,C 180,E1 -27430.991,E2 -27430.991} C_VEL
LIN {X 0,Y 84.226,Z 540.995,A -85,B 0,C 180,E1 -27440.41,E2 -27440.41} C_VEL
LIN {X 0,Y 83.965,Z 540.046,A -85,B 0,C 180,E1 -27445.215,E2 -27445.215} C_VEL
LIN {X 0,Y 84.132,Z 538.661,A -85,B 0,C 180,E1 -27450.016,E2 -27450.016} C_VEL
LIN {X 0,Y 84.115,Z 535.69,A -85,B 0,C 180,E1 -27457.215,E2 -27457.215} C_VEL
LIN {X 0,Y 85.02,Z 531.609,A -85,B 0,C 180,E1 -27464.373,E2 -27464.373} C_VEL
LIN {X 0,Y 87.438,Z 525.281,A -85,B 0,C 180,E1 -27472.459,E2 -27472.459} C_VEL
LIN {X 0,Y 90.783,Z 518.36,A -85,B 0,C 180,E1 -27478.951,E2 -27478.951} C_VEL
LIN {X 0,Y 94.3,Z 511.258,A -85,B 0,C 180,E1 -27483.998,E2 -27483.998} C_VEL
LIN {X 0,Y 98.439,Z 502.879,A -85,B 0,C 180,E1 -27488.542,E2 -27488.542} C_VEL
LIN {X 0,Y 103.386,Z 492.103,A -85,B 0,C 180,E1 -27492.84,E2 -27492.84} C_VEL
LIN {X 0,Y 107.632,Z 481.644,A -85,B 0,C 180,E1 -27495.925,E2 -27495.925} C_VEL
LIN {X 0,Y 111.584,Z 470.18,A -85,B 0,C 180,E1 -27498.425,E2 -27498.425} C_VEL
LIN {X 0,Y 114.855,Z 458.44,A -85,B 0,C 180,E1 -27500.251,E2 -27500.251} C_VEL
LIN {X 0,Y 117.642,Z 445.095,A -85,B 0,C 180,E1 -27501.673,E2 -27501.673} C_VEL
LIN {X 0,Y 119.274,Z 432.314,A -85,B 0,C 180,E1 -27502.547,E2 -27502.547} C_VEL
LIN {X 0,Y 121.913,Z 402.898,A -85,B 0,C 180,E1 -27504.054,E2 -27504.054} C_VEL
LIN {X 0,Y 118.966,Z 393.121,A -85,B 0,C 180,E1 -27506.326,E2 -27506.326} C_VEL
LIN {X 0,Y 117.678,Z 389.959,A -85,B 0,C 180,E1 -27507.266,E2 -27507.266} C_VEL
LIN {X 0,Y 115.053,Z 386.01,A -85,B 0,C 180,E1 -27509.018,E2 -27509.018} C_VEL
LIN {X 0,Y 106.147,Z 376.426,A -85,B 0,C 180,E1 -27515.604,E2 -27515.604} C_VEL
LIN {X 0,Y 104.552,Z 373.883,A -85,B 0,C 180,E1 -27517.096,E2 -27517.096} C_VEL
LIN {X 0,Y 101.367,Z 368.792,A -85,B 0,C 180,E1 -27520.42,E2 -27520.42} C_VEL
LIN {X 0,Y 99.222,Z 365.385,A -85,B 0,C 180,E1 -27522.971,E2 -27522.971} C_VEL
LIN {X 0,Y 96.803,Z 361.787,A -85,B 0,C 180,E1 -27526.105,E2 -27526.105} C_VEL
LIN {X 0,Y 94.44,Z 358.419,A -85,B 0,C 180,E1 -27529.656,E2 -27529.656} C_VEL
LIN {X 0,Y 93.847,Z 357.289,A -85,B 0,C 180,E1 -27530.719,E2 -27530.719} C_VEL
LIN {X 0,Y 91.514,Z 354.529,A -85,B 0,C 180,E1 -27535.078,E2 -27535.078} C_VEL
LIN {X 0,Y 90.412,Z 352.153,A -85,B 0,C 180,E1 -27537.826,E2 -27537.826} C_VEL
LIN {X 0,Y 88.383,Z 350.83,A -85,B 0,C 180,E1 -27543.419,E2 -27543.419} C_VEL
LIN {X 0,Y 86.845,Z 349.284,A -85,B 0,C 180,E1 -27551.256,E2 -27551.256} C_VEL
LIN {X 0,Y 86.567,Z 349.276,A -85,B 0,C 180,E1 -27556.627,E2 -27556.627} C_VEL
LIN {X 0,Y 87.337,Z 350.666,A -85,B 0,C 180,E1 -27565.379,E2 -27565.379} C_VEL
LIN {X 0,Y 90.102,Z 352.694,A -85,B 0,C 180,E1 -27574.372,E2 -27574.372} C_VEL
LIN {X 0,Y 91.975,Z 356.116,A -85,B 0,C 180,E1 -27578.809,E2 -27578.809} C_VEL
LIN {X 0,Y 93.981,Z 358.042,A -85,B 0,C 180,E1 -27582.302,E2 -27582.302} C_VEL
LIN {X 0,Y 96.421,Z 361.656,A -85,B 0,C 180,E1 -27586.123,E2 -27586.123} C_VEL
LIN {X 0,Y 97.436,Z 362.932,A -85,B 0,C 180,E1 -27587.483,E2 -27587.483} C_VEL
LIN {X 0,Y 100.806,Z 367.87,A -85,B 0,C 180,E1 -27591.602,E2 -27591.602} C_VEL
LIN {X 0,Y 104.625,Z 374.003,A -85,B 0,C 180,E1 -27595.653,E2 -27595.653} C_VEL
LIN {X 0,Y 109.155,Z 381.953,A -85,B 0,C 180,E1 -27599.765,E2 -27599.765} C_VEL
LIN {X 0,Y 114.98,Z 393.64,A -85,B 0,C 180,E1 -27604.423,E2 -27604.423} C_VEL
LIN {X 0,Y 116.949,Z 398.585,A -85,B 0,C 180,E1 -27605.909,E2 -27605.909} C_VEL
LIN {X 0,Y 113.453,Z 433.397,A -85,B 0,C 180,E1 -27607.777,E2 -27607.777} C_VEL
LIN {X 0,Y 111.022,Z 447.368,A -85,B 0,C 180,E1 -27609.129,E2 -27609.129} C_VEL
LIN {X 0,Y 107.812,Z 459.983,A -85,B 0,C 180,E1 -27610.966,E2 -27610.966} C_VEL
LIN {X 0,Y 104.068,Z 471.479,A -85,B 0,C 180,E1 -27613.309,E2 -27613.309} C_VEL
LIN {X 0,Y 99.844,Z 482.11,A -85,B 0,C 180,E1 -27616.204,E2 -27616.204} C_VEL
LIN {X 0,Y 95.31,Z 492.176,A -85,B 0,C 180,E1 -27619.901,E2 -27619.901} C_VEL
LIN {X 0,Y 90.415,Z 501.921,A -85,B 0,C 180,E1 -27624.781,E2 -27624.781} C_VEL
LIN {X 0,Y 86.295,Z 509.682,A -85,B 0,C 180,E1 -27629.985,E2 -27629.985} C_VEL
LIN {X 0,Y 82.634,Z 516.566,A -85,B 0,C 180,E1 -27636.086,E2 -27636.086} C_VEL
LIN {X 0,Y 79.505,Z 522.835,A -85,B 0,C 180,E1 -27643.501,E2 -27643.501} C_VEL
LIN {X 0,Y 77.504,Z 527.695,A -85,B 0,C 180,E1 -27651.247,E2 -27651.247} C_VEL
LIN {X 0,Y 76.342,Z 531.831,A -85,B 0,C 180,E1 -27660.397,E2 -27660.397} C_VEL
LIN {X 0,Y 76.924,Z 534.642,A -85,B 0,C 180,E1 -27669.732,E2 -27669.732} C_VEL
LIN {X 0,Y 78.32,Z 535.835,A -85,B 0,C 180,E1 -27675.851,E2 -27675.851} C_VEL
LIN {X 0,Y 80.738,Z 536.498,A -85,B 0,C 180,E1 -27682.459,E2 -27682.459} C_VEL
LIN {X 0,Y 85.154,Z 536.362,A -85,B 0,C 180,E1 -27690.317,E2 -27690.317} C_VEL
LIN {X 0,Y 91.193,Z 535.022,A -85,B 0,C 180,E1 -27697.592,E2 -27697.592} C_VEL
LIN {X 0,Y 97.695,Z 532.735,A -85,B 0,C 180,E1 -27703.276,E2 -27703.276} C_VEL
LIN {X 0,Y 105.462,Z 529.172,A -85,B 0,C 180,E1 -27708.468,E2 -27708.468} C_VEL
LIN {X 0,Y 113.983,Z 524.277,A -85,B 0,C 180,E1 -27712.916,E2 -27712.916} C_VEL
LIN {X 0,Y 123.027,Z 517.905,A -85,B 0,C 180,E1 -27716.725,E2 -27716.725} C_VEL
LIN {X 0,Y 131.907,Z 510.397,A -85,B 0,C 180,E1 -27719.79,E2 -27719.79} C_VEL
LIN {X 0,Y 140.64,Z 501.517,A -85,B 0,C 180,E1 -27722.294,E2 -27722.294} C_VEL
LIN {X 0,Y 148.714,Z 491.637,A -85,B 0,C 180,E1 -27724.258,E2 -27724.258} C_VEL
LIN {X 0,Y 155.363,Z 481.78,A -85,B 0,C 180,E1 -27725.746,E2 -27725.746} C_VEL
LIN {X 0,Y 161.016,Z 471.619,A -85,B 0,C 180,E1 -27726.892,E2 -27726.892} C_VEL
LIN {X 0,Y 166.17,Z 459.971,A -85,B 0,C 180,E1 -27727.886,E2 -27727.886} C_VEL
LIN {X 0,Y 170.421,Z 447.099,A -85,B 0,C 180,E1 -27728.699,E2 -27728.699} C_VEL
LIN {X 0,Y 172.576,Z 438.249,A -85,B 0,C 180,E1 -27729.086,E2 -27729.086} C_VEL
LIN {X 0,Y 172.202,Z 436.774,A -85,B 0,C 180,E1 -27730.996,E2 -27730.996} C_VEL
LIN {X 0,Y 171.78,Z 435.948,A -85,B 0,C 180,E1 -27734.21,E2 -27734.21} C_VEL
LIN {X 0,Y 171.773,Z 436.14,A -85,B 0,C 180,E1 -27737.276,E2 -27737.276} C_VEL
LIN {X 0,Y 172.112,Z 437.084,A -85,B 0,C 180,E1 -27740.119,E2 -27740.119} C_VEL
LIN {X 0,Y 172.42,Z 439.737,A -85,B 0,C 180,E1 -27742.466,E2 -27742.466} C_VEL
LIN {X 0,Y 169.214,Z 452.316,A -85,B 0,C 180,E1 -27742.991,E2 -27742.991} C_VEL
LIN {X 0,Y 164.74,Z 464.597,A -85,B 0,C 180,E1 -27743.65,E2 -27743.65} C_VEL
LIN {X 0,Y 159.255,Z 476.174,A -85,B 0,C 180,E1 -27744.496,E2 -27744.496} C_VEL
LIN {X 0,Y 152.945,Z 486.939,A -85,B 0,C 180,E1 -27745.634,E2 -27745.634} C_VEL
LIN {X 0,Y 145.931,Z 496.786,A -85,B 0,C 180,E1 -27747.034,E2 -27747.034} C_VEL
LIN {X 0,Y 136.861,Z 507.338,A -85,B 0,C 180,E1 -27749.221,E2 -27749.221} C_VEL
LIN {X 0,Y 127.999,Z 515.912,A -85,B 0,C 180,E1 -27751.699,E2 -27751.699} C_VEL
LIN {X 0,Y 119.611,Z 522.807,A -85,B 0,C 180,E1 -27754.679,E2 -27754.679} C_VEL
LIN {X 0,Y 111.519,Z 528.412,A -85,B 0,C 180,E1 -27758.047,E2 -27758.047} C_VEL
LIN {X 0,Y 103.993,Z 532.888,A -85,B 0,C 180,E1 -27762.002,E2 -27762.002} C_VEL
LIN {X 0,Y 95.006,Z 537.283,A -85,B 0,C 180,E1 -27768.281,E2 -27768.281} C_VEL
LIN {X 0,Y 87.331,Z 540.113,A -85,B 0,C 180,E1 -27775.735,E2 -27775.735} C_VEL
LIN {X 0,Y 81.512,Z 541.375,A -85,B 0,C 180,E1 -27784.482,E2 -27784.482} C_VEL
LIN {X 0,Y 78.095,Z 541.2,A -85,B 0,C 180,E1 -27794.356,E2 -27794.356} C_VEL
LIN {X 0,Y 77.218,Z 540.556,A -85,B 0,C 180,E1 -27799.53,E2 -27799.53} C_VEL
LIN {X 0,Y 76.913,Z 539.495,A -85,B 0,C 180,E1 -27804.775,E2 -27804.775} C_VEL
LIN {X 0,Y 77.049,Z 538.028,A -85,B 0,C 180,E1 -27810.017,E2 -27810.017} C_VEL
LIN {X 0,Y 77.084,Z 534.912,A -85,B 0,C 180,E1 -27817.877,E2 -27817.877} C_VEL
LIN {X 0,Y 78.134,Z 530.674,A -85,B 0,C 180,E1 -27825.671,E2 -27825.671} C_VEL
LIN {X 0,Y 80.908,Z 524.189,A -85,B 0,C 180,E1 -27834.385,E2 -27834.385} C_VEL
LIN {X 0,Y 84.611,Z 517.038,A -85,B 0,C 180,E1 -27841.29,E2 -27841.29} C_VEL
LIN {X 0,Y 89.352,Z 508.082,A -85,B 0,C 180,E1 -27847.574,E2 -27847.574} C_VEL
LIN {X 0,Y 94.046,Z 498.894,A -85,B 0,C 180,E1 -27852.281,E2 -27852.281} C_VEL
LIN {X 0,Y 98.786,Z 488.711,A -85,B 0,C 180,E1 -27856.097,E2 -27856.097} C_VEL
LIN {X 0,Y 103.422,Z 477.497,A -85,B 0,C 180,E1 -27859.127,E2 -27859.127} C_VEL
LIN {X 0,Y 107.011,Z 466.888,A -85,B 0,C 180,E1 -27861.266,E2 -27861.266} C_VEL
LIN {X 0,Y 110.437,Z 454.231,A -85,B 0,C 180,E1 -27863.092,E2 -27863.092} C_VEL
LIN {X 0,Y 112.933,Z 441.293,A -85,B 0,C 180,E1 -27864.31,E2 -27864.31} C_VEL
LIN {X 0,Y 115.202,Z 420.655,A -85,B 0,C 180,E1 -27865.474,E2 -27865.474} C_VEL
LIN {X 0,Y 116.637,Z 404.546,A -85,B 0,C 180,E1 -27866.345,E2 -27866.345} C_VEL
LIN {X 0,Y 112.719,Z 391.707,A -85,B 0,C 180,E1 -27869.668,E2 -27869.668} C_VEL
LIN {X 0,Y 109.166,Z 382.313,A -85,B 0,C 180,E1 -27872.849,E2 -27872.849} C_VEL
LIN {X 0,Y 104.552,Z 373.883,A -85,B 0,C 180,E1 -27877.096,E2 -27877.096} C_VEL
LIN {X 0,Y 102.906,Z 371.794,A -85,B 0,C 180,E1 -27878.682,E2 -27878.682} C_VEL
LIN {X 0,Y 100.973,Z 370.596,A -85,B 0,C 180,E1 -27880.51,E2 -27880.51} C_VEL
LIN {X 0,Y 95.17,Z 368.578,A -85,B 0,C 180,E1 -27886.736,E2 -27886.736} C_VEL
LIN {X 0,Y 94.632,Z 368.164,A -85,B 0,C 180,E1 -27887.456,E2 -27887.456} C_VEL
LIN {X 0,Y 92.185,Z 364.4,A -85,B 0,C 180,E1 -27891.556,E2 -27891.556} C_VEL
LIN {X 0,Y 91.259,Z 363.158,A -85,B 0,C 180,E1 -27893.328,E2 -27893.328} C_VEL
LIN {X 0,Y 89.193,Z 359.835,A -85,B 0,C 180,E1 -27897.999,E2 -27897.999} C_VEL
LIN {X 0,Y 88.745,Z 358.798,A -85,B 0,C 180,E1 -27899.33,E2 -27899.33} C_VEL
LIN {X 0,Y 85.887,Z 356.396,A -85,B 0,C 180,E1 -27910.846,E2 -27910.846} C_VEL
LIN {X 0,Y 85.572,Z 356.34,A -85,B 0,C 180,E1 -27916.826,E2 -27916.826} C_VEL
LIN {X 0,Y 86.379,Z 357.831,A -85,B 0,C 180,E1 -27925.681,E2 -27925.681} C_VEL
LIN {X 0,Y 88.564,Z 359.529,A -85,B 0,C 180,E1 -27933.173,E2 -27933.173} C_VEL
LIN {X 0,Y 90.485,Z 362.966,A -85,B 0,C 180,E1 -27938.046,E2 -27938.046} C_VEL
LIN {X 0,Y 92.051,Z 364.604,A -85,B 0,C 180,E1 -27940.943,E2 -27940.943} C_VEL
LIN {X 0,Y 94.547,Z 368.325,A -85,B 0,C 180,E1 -27945.148,E2 -27945.148} C_VEL
LIN {X 0,Y 98.19,Z 373.966,A -85,B 0,C 180,E1 -27950.084,E2 -27950.084} C_VEL
LIN {X 0,Y 102.162,Z 380.807,A -85,B 0,C 180,E1 -27954.644,E2 -27954.644} C_VEL
LIN {X 0,Y 105.913,Z 387.897,A -85,B 0,C 180,E1 -27958.344,E2 -27958.344} C_VEL
LIN {X 0,Y 110.814,Z 398.153,A -85,B 0,C 180,E1 -27962.611,E2 -27962.611} C_VEL
LIN {X 0,Y 111.829,Z 400.881,A -85,B 0,C 180,E1 -27963.479,E2 -27963.479} C_VEL
LIN {X 0,Y 108.379,Z 433.395,A -85,B 0,C 180,E1 -27965.211,E2 -27965.211} C_VEL
LIN {X 0,Y 105.913,Z 447.072,A -85,B 0,C 180,E1 -27966.526,E2 -27966.526} C_VEL
LIN {X 0,Y 102.555,Z 459.864,A -85,B 0,C 180,E1 -27968.374,E2 -27968.374} C_VEL
LIN {X 0,Y 98.626,Z 471.43,A -85,B 0,C 180,E1 -27970.744,E2 -27970.744} C_VEL
LIN {X 0,Y 94.13,Z 482.228,A -85,B 0,C 180,E1 -27973.727,E2 -27973.727} C_VEL
LIN {X 0,Y 88.784,Z 493.344,A -85,B 0,C 180,E1 -27977.993,E2 -27977.993} C_VEL
LIN {X 0,Y 83.795,Z 502.679,A -85,B 0,C 180,E1 -27982.991,E2 -27982.991} C_VEL
LIN {X 0,Y 79.308,Z 510.576,A -85,B 0,C 180,E1 -27988.714,E2 -27988.714} C_VEL
LIN {X 0,Y 75.453,Z 517.363,A -85,B 0,C 180,E1 -27995.327,E2 -27995.327} C_VEL
LIN {X 0,Y 72.257,Z 523.518,A -85,B 0,C 180,E1 -28003.432,E2 -28003.432} C_VEL
LIN {X 0,Y 70.505,Z 527.479,A -85,B 0,C 180,E1 -28010.398,E2 -28010.398} C_VEL
LIN {X 0,Y 69.256,Z 531.76,A -85,B 0,C 180,E1 -28020.466,E2 -28020.466} C_VEL
LIN {X 0,Y 69.475,Z 533.85,A -85,B 0,C 180,E1 -28027.343,E2 -28027.343} C_VEL
LIN {X 0,Y 71.183,Z 535.777,A -85,B 0,C 180,E1 -28036.281,E2 -28036.281} C_VEL
LIN {X 0,Y 75.408,Z 536.851,A -85,B 0,C 180,E1 -28046.975,E2 -28046.975} C_VEL
LIN {X 0,Y 79.797,Z 536.639,A -85,B 0,C 180,E1 -28053.873,E2 -28053.873} C_VEL
LIN {X 0,Y 86.158,Z 535.387,A -85,B 0,C 180,E1 -28060.956,E2 -28060.956} C_VEL
LIN {X 0,Y 93.725,Z 532.983,A -85,B 0,C 180,E1 -28067.034,E2 -28067.034} C_VEL
LIN {X 0,Y 102.075,Z 529.415,A -85,B 0,C 180,E1 -28072.085,E2 -28072.085} C_VEL
LIN {X 0,Y 111.122,Z 524.491,A -85,B 0,C 180,E1 -28076.374,E2 -28076.374} C_VEL
LIN {X 0,Y 120.775,Z 518.012,A -85,B 0,C 180,E1 -28080,E2 -28080} C_VEL
LIN {X 0,Y 128.645,Z 511.7,A -85,B 0,C 180,E1 -28082.504,E2 -28082.504} C_VEL
LIN {X 0,Y 137.502,Z 503.293,A -85,B 0,C 180,E1 -28084.831,E2 -28084.831} C_VEL
LIN {X 0,Y 145.633,Z 493.996,A -85,B 0,C 180,E1 -28086.64,E2 -28086.64} C_VEL
LIN {X 0,Y 152.758,Z 484.065,A -85,B 0,C 180,E1 -28088.112,E2 -28088.112} C_VEL
LIN {X 0,Y 159.206,Z 473.089,A -85,B 0,C 180,E1 -28089.296,E2 -28089.296} C_VEL
LIN {X 0,Y 164.867,Z 460.93,A -85,B 0,C 180,E1 -28090.275,E2 -28090.275} C_VEL
LIN {X 0,Y 169.323,Z 448.011,A -85,B 0,C 180,E1 -28091.041,E2 -28091.041} C_VEL
LIN {X 0,Y 170.516,Z 443.633,A -85,B 0,C 180,E1 -28091.261,E2 -28091.261} C_VEL
LIN {X 0,Y 170.198,Z 442.853,A -85,B 0,C 180,E1 -28094.345,E2 -28094.345} C_VEL
LIN {X 0,Y 170.224,Z 443.159,A -85,B 0,C 180,E1 -28097.587,E2 -28097.587} C_VEL
LIN {X 0,Y 170.426,Z 443.818,A -85,B 0,C 180,E1 -28099.576,E2 -28099.576} C_VEL
LIN {X 0,Y 170.413,Z 444.586,A -85,B 0,C 180,E1 -28100.287,E2 -28100.287} C_VEL
LIN {X 0,Y 166.642,Z 456.999,A -85,B 0,C 180,E1 -28100.808,E2 -28100.808} C_VEL
LIN {X 0,Y 161.937,Z 468.426,A -85,B 0,C 180,E1 -28101.411,E2 -28101.411} C_VEL
LIN {X 0,Y 155.693,Z 480.266,A -85,B 0,C 180,E1 -28102.307,E2 -28102.307} C_VEL
LIN {X 0,Y 148.436,Z 491.358,A -85,B 0,C 180,E1 -28103.49,E2 -28103.49} C_VEL
LIN {X 0,Y 141.337,Z 500.354,A -85,B 0,C 180,E1 -28104.871,E2 -28104.871} C_VEL
LIN {X 0,Y 132.054,Z 510.114,A -85,B 0,C 180,E1 -28106.975,E2 -28106.975} C_VEL
LIN {X 0,Y 122.932,Z 518.059,A -85,B 0,C 180,E1 -28109.355,E2 -28109.355} C_VEL
LIN {X 0,Y 115.742,Z 523.492,A -85,B 0,C 180,E1 -28111.806,E2 -28111.806} C_VEL
LIN {X 0,Y 107.299,Z 528.911,A -85,B 0,C 180,E1 -28115.068,E2 -28115.068} C_VEL
LIN {X 0,Y 99.382,Z 533.211,A -85,B 0,C 180,E1 -28118.958,E2 -28118.958} C_VEL
LIN {X 0,Y 89.825,Z 537.426,A -85,B 0,C 180,E1 -28125.262,E2 -28125.262} C_VEL
LIN {X 0,Y 81.537,Z 540.027,A -85,B 0,C 180,E1 -28132.913,E2 -28132.913} C_VEL
LIN {X 0,Y 75.139,Z 541.143,A -85,B 0,C 180,E1 -28142.139,E2 -28142.139} C_VEL
LIN {X 0,Y 71.28,Z 540.808,A -85,B 0,C 180,E1 -28152.815,E2 -28152.815} C_VEL
LIN {X 0,Y 69.849,Z 538.925,A -85,B 0,C 180,E1 -28164.245,E2 -28164.245} C_VEL
LIN {X 0,Y 69.956,Z 537.395,A -85,B 0,C 180,E1 -28170.019,E2 -28170.019} C_VEL
LIN {X 0,Y 70.058,Z 534.135,A -85,B 0,C 180,E1 -28178.673,E2 -28178.673} C_VEL
LIN {X 0,Y 71.307,Z 529.742,A -85,B 0,C 180,E1 -28187.216,E2 -28187.216} C_VEL
LIN {X 0,Y 73.897,Z 524.106,A -85,B 0,C 180,E1 -28195.357,E2 -28195.357} C_VEL
LIN {X 0,Y 77.829,Z 517.019,A -85,B 0,C 180,E1 -28202.824,E2 -28202.824} C_VEL
LIN {X 0,Y 82.867,Z 508.115,A -85,B 0,C 180,E1 -28209.517,E2 -28209.517} C_VEL
LIN {X 0,Y 88.306,Z 498.083,A -85,B 0,C 180,E1 -28214.874,E2 -28214.874} C_VEL
LIN {X 0,Y 93.408,Z 487.626,A -85,B 0,C 180,E1 -28218.815,E2 -28218.815} C_VEL
LIN {X 0,Y 98.264,Z 476.213,A -85,B 0,C 180,E1 -28221.898,E2 -28221.898} C_VEL
LIN {X 0,Y 102.395,Z 464.353,A -85,B 0,C 180,E1 -28224.187,E2 -28224.187} C_VEL
LIN {X 0,Y 105.989,Z 450.645,A -85,B 0,C 180,E1 -28225.998,E2 -28225.998} C_VEL
LIN {X 0,Y 108.397,Z 437.363,A -85,B 0,C 180,E1 -28227.113,E2 -28227.113} C_VEL
LIN {X 0,Y 111.55,Z 406.53,A -85,B 0,C 180,E1 -28228.746,E2 -28228.746} C_VEL
LIN {X 0,Y 107.92,Z 394.158,A -85,B 0,C 180,E1 -28232.262,E2 -28232.262} C_VEL
LIN {X 0,Y 105.114,Z 386.474,A -85,B 0,C 180,E1 -28235.069,E2 -28235.069} C_VEL
LIN {X 0,Y 100.63,Z 378.021,A -85,B 0,C 180,E1 -28239.704,E2 -28239.704} C_VEL
LIN {X 0,Y 96.58,Z 371.312,A -85,B 0,C 180,E1 -28244.676,E2 -28244.676} C_VEL
LIN {X 0,Y 94.632,Z 368.164,A -85,B 0,C 180,E1 -28247.456,E2 -28247.456} C_VEL
LIN {X 0,Y 91.715,Z 366.256,A -85,B 0,C 180,E1 -28251.841,E2 -28251.841} C_VEL
LIN {X 0,Y 87.95,Z 365.198,A -85,B 0,C 180,E1 -28259.071,E2 -28259.071} C_VEL
LIN {X 0,Y 85.495,Z 364.321,A -85,B 0,C 180,E1 -28266.847,E2 -28266.847} C_VEL
LIN {X 0,Y 84.755,Z 363.304,A -85,B 0,C 180,E1 -28272.15,E2 -28272.15} C_VEL
LIN {X 0,Y 84.622,Z 363.661,A -85,B 0,C 180,E1 -28279.403,E2 -28279.403} C_VEL
LIN {X 0,Y 87.077,Z 366.313,A -85,B 0,C 180,E1 -28291.938,E2 -28291.938} C_VEL
LIN {X 0,Y 89.032,Z 369.853,A -85,B 0,C 180,E1 -28297.305,E2 -28297.305} C_VEL
LIN {X 0,Y 90.122,Z 371.138,A -85,B 0,C 180,E1 -28299.502,E2 -28299.502} C_VEL
LIN {X 0,Y 92.938,Z 375.682,A -85,B 0,C 180,E1 -28304.579,E2 -28304.579} C_VEL
LIN {X 0,Y 95.504,Z 379.872,A -85,B 0,C 180,E1 -28308.345,E2 -28308.345} C_VEL
LIN {X 0,Y 99.237,Z 386.64,A -85,B 0,C 180,E1 -28313.015,E2 -28313.015} C_VEL
LIN {X 0,Y 102.932,Z 394.191,A -85,B 0,C 180,E1 -28317.03,E2 -28317.03} C_VEL
LIN {X 0,Y 106.773,Z 402.788,A -85,B 0,C 180,E1 -28320.678,E2 -28320.678} C_VEL
LIN {X 0,Y 106.94,Z 403.229,A -85,B 0,C 180,E1 -28320.836,E2 -28320.836} C_VEL
LIN {X 0,Y 103.494,Z 433.749,A -85,B 0,C 180,E1 -28322.43,E2 -28322.43} C_VEL
LIN {X 0,Y 100.943,Z 447.272,A -85,B 0,C 180,E1 -28323.732,E2 -28323.732} C_VEL
LIN {X 0,Y 97.535,Z 459.715,A -85,B 0,C 180,E1 -28325.51,E2 -28325.51} C_VEL
LIN {X 0,Y 93.384,Z 471.359,A -85,B 0,C 180,E1 -28327.882,E2 -28327.882} C_VEL
LIN {X 0,Y 88.581,Z 482.359,A -85,B 0,C 180,E1 -28330.953,E2 -28330.953} C_VEL
LIN {X 0,Y 82.979,Z 493.369,A -85,B 0,C 180,E1 -28335.265,E2 -28335.265} C_VEL
LIN {X 0,Y 77.322,Z 503.282,A -85,B 0,C 180,E1 -28340.831,E2 -28340.831} C_VEL
LIN {X 0,Y 72.367,Z 511.408,A -85,B 0,C 180,E1 -28347.199,E2 -28347.199} C_VEL
LIN {X 0,Y 68.282,Z 518.132,A -85,B 0,C 180,E1 -28354.456,E2 -28354.456} C_VEL
LIN {X 0,Y 64.998,Z 524.104,A -85,B 0,C 180,E1 -28363.31,E2 -28363.31} C_VEL
LIN {X 0,Y 62.949,Z 528.683,A -85,B 0,C 180,E1 -28372.571,E2 -28372.571} C_VEL
LIN {X 0,Y 62.18,Z 532.811,A -85,B 0,C 180,E1 -28384.383,E2 -28384.383} C_VEL
LIN {X 0,Y 62.99,Z 534.748,A -85,B 0,C 180,E1 -28391.992,E2 -28391.992} C_VEL
LIN {X 0,Y 64.775,Z 536.086,A -85,B 0,C 180,E1 -28399.383,E2 -28399.383} C_VEL
LIN {X 0,Y 69.005,Z 537.077,A -85,B 0,C 180,E1 -28409.387,E2 -28409.387} C_VEL
LIN {X 0,Y 75.418,Z 536.861,A -85,B 0,C 180,E1 -28418.67,E2 -28418.67} C_VEL
LIN {X 0,Y 81.891,Z 535.667,A -85,B 0,C 180,E1 -28425.08,E2 -28425.08} C_VEL
LIN {X 0,Y 90.07,Z 533.277,A -85,B 0,C 180,E1 -28431.022,E2 -28431.022} C_VEL
LIN {X 0,Y 99.095,Z 529.673,A -85,B 0,C 180,E1 -28435.933,E2 -28435.933} C_VEL
LIN {X 0,Y 108.69,Z 524.746,A -85,B 0,C 180,E1 -28440,E2 -28440} C_VEL
LIN {X 0,Y 118.851,Z 518.242,A -85,B 0,C 180,E1 -28443.39,E2 -28443.39} C_VEL
LIN {X 0,Y 127.099,Z 511.863,A -85,B 0,C 180,E1 -28445.693,E2 -28445.693} C_VEL
LIN {X 0,Y 136.364,Z 503.309,A -85,B 0,C 180,E1 -28447.849,E2 -28447.849} C_VEL
LIN {X 0,Y 145.198,Z 493.335,A -85,B 0,C 180,E1 -28449.606,E2 -28449.606} C_VEL
LIN {X 0,Y 152.55,Z 483.226,A -85,B 0,C 180,E1 -28450.906,E2 -28450.906} C_VEL
LIN {X 0,Y 159.276,Z 471.834,A -85,B 0,C 180,E1 -28451.989,E2 -28451.989} C_VEL
LIN {X 0,Y 164.991,Z 459.281,A -85,B 0,C 180,E1 -28452.87,E2 -28452.87} C_VEL
LIN {X 0,Y 168.317,Z 449.858,A -85,B 0,C 180,E1 -28453.378,E2 -28453.378} C_VEL
LIN {X 0,Y 168.267,Z 449.849,A -85,B 0,C 180,E1 -28457,E2 -28457} C_VEL
LIN {X 0,Y 168.323,Z 450.144,A -85,B 0,C 180,E1 -28458.067,E2 -28458.067} C_VEL
LIN {X 0,Y 163.92,Z 462.374,A -85,B 0,C 180,E1 -28458.594,E2 -28458.594} C_VEL
LIN {X 0,Y 158.162,Z 474.364,A -85,B 0,C 180,E1 -28459.257,E2 -28459.257} C_VEL
LIN {X 0,Y 151.555,Z 485.329,A -85,B 0,C 180,E1 -28460.144,E2 -28460.144} C_VEL
LIN {X 0,Y 144.173,Z 495.355,A -85,B 0,C 180,E1 -28461.241,E2 -28461.241} C_VEL
LIN {X 0,Y 135.353,Z 505.272,A -85,B 0,C 180,E1 -28462.868,E2 -28462.868} C_VEL
LIN {X 0,Y 125.891,Z 514.052,A -85,B 0,C 180,E1 -28464.916,E2 -28464.916} C_VEL
LIN {X 0,Y 118.161,Z 520.099,A -85,B 0,C 180,E1 -28466.885,E2 -28466.885} C_VEL
LIN {X 0,Y 109.232,Z 526.076,A -85,B 0,C 180,E1 -28469.736,E2 -28469.736} C_VEL
LIN {X 0,Y 100.563,Z 530.898,A -85,B 0,C 180,E1 -28473.034,E2 -28473.034} C_VEL
LIN {X 0,Y 89.859,Z 535.757,A -85,B 0,C 180,E1 -28478.574,E2 -28478.574} C_VEL
LIN {X 0,Y 80.265,Z 538.927,A -85,B 0,C 180,E1 -28485.561,E2 -28485.561} C_VEL
LIN {X 0,Y 72.2,Z 540.61,A -85,B 0,C 180,E1 -28494.29,E2 -28494.29} C_VEL
LIN {X 0,Y 68.921,Z 540.908,A -85,B 0,C 180,E1 -28499.37,E2 -28499.37} C_VEL
LIN {X 0,Y 64.502,Z 540.361,A -85,B 0,C 180,E1 -28510.944,E2 -28510.944} C_VEL
LIN {X 0,Y 62.808,Z 538.337,A -85,B 0,C 180,E1 -28523.597,E2 -28523.597} C_VEL
LIN {X 0,Y 62.89,Z 536.729,A -85,B 0,C 180,E1 -28530.021,E2 -28530.021} C_VEL
LIN {X 0,Y 63.041,Z 533.326,A -85,B 0,C 180,E1 -28539.647,E2 -28539.647} C_VEL
LIN {X 0,Y 64.521,Z 528.772,A -85,B 0,C 180,E1 -28549.093,E2 -28549.093} C_VEL
LIN {X 0,Y 68.182,Z 521.815,A -85,B 0,C 180,E1 -28559.335,E2 -28559.335} C_VEL
LIN {X 0,Y 72.805,Z 514.251,A -85,B 0,C 180,E1 -28567.128,E2 -28567.128} C_VEL
LIN {X 0,Y 78.192,Z 505.357,A -85,B 0,C 180,E1 -28573.557,E2 -28573.557} C_VEL
LIN {X 0,Y 84.062,Z 494.888,A -85,B 0,C 180,E1 -28578.822,E2 -28578.822} C_VEL
LIN {X 0,Y 89.518,Z 483.913,A -85,B 0,C 180,E1 -28582.666,E2 -28582.666} C_VEL
LIN {X 0,Y 94.01,Z 473.2,A -85,B 0,C 180,E1 -28585.338,E2 -28585.338} C_VEL
LIN {X 0,Y 98.38,Z 460.445,A -85,B 0,C 180,E1 -28587.568,E2 -28587.568} C_VEL
LIN {X 0,Y 101.614,Z 447.84,A -85,B 0,C 180,E1 -28589.061,E2 -28589.061} C_VEL
LIN {X 0,Y 103.932,Z 433.874,A -85,B 0,C 180,E1 -28590.101,E2 -28590.101} C_VEL
LIN {X 0,Y 106.636,Z 408.326,A -85,B 0,C 180,E1 -28591.422,E2 -28591.422} C_VEL
LIN {X 0,Y 103.643,Z 397.705,A -85,B 0,C 180,E1 -28594.69,E2 -28594.69} C_VEL
LIN {X 0,Y 101.296,Z 390.932,A -85,B 0,C 180,E1 -28597.321,E2 -28597.321} C_VEL
LIN {X 0,Y 97.226,Z 382.781,A -85,B 0,C 180,E1 -28602.123,E2 -28602.123} C_VEL
LIN {X 0,Y 93.59,Z 376.552,A -85,B 0,C 180,E1 -28607.109,E2 -28607.109} C_VEL
LIN {X 0,Y 91.999,Z 373.893,A -85,B 0,C 180,E1 -28609.708,E2 -28609.708} C_VEL
LIN {X 0,Y 89.7,Z 369.958,A -85,B 0,C 180,E1 -28614.196,E2 -28614.196} C_VEL
LIN {X 0,Y 87.666,Z 366.648,A -85,B 0,C 180,E1 -28619.152,E2 -28619.152} C_VEL
LIN {X 0,Y 87.142,Z 365.479,A -85,B 0,C 180,E1 -28620.867,E2 -28620.867} C_VEL
LIN {X 0,Y 85.495,Z 364.321,A -85,B 0,C 180,E1 -28626.847,E2 -28626.847} C_VEL
LIN {X 0,Y 84.982,Z 364.24,A -85,B 0,C 180,E1 -28629.465,E2 -28629.465} C_VEL
LIN {X 0,Y 84.557,Z 364.846,A -85,B 0,C 180,E1 -28632.082,E2 -28632.082} C_VEL
LIN {X 0,Y 84.023,Z 367.321,A -85,B 0,C 180,E1 -28637.222,E2 -28637.222} C_VEL
LIN {X 0,Y 84.266,Z 371.595,A -85,B 0,C 180,E1 -28645.016,E2 -28645.016} C_VEL
LIN {X 0,Y 84.794,Z 372.426,A -85,B 0,C 180,E1 -28647.68,E2 -28647.68} C_VEL
LIN {X 0,Y 85.629,Z 373.101,A -85,B 0,C 180,E1 -28650.661,E2 -28650.661} C_VEL
LIN {X 0,Y 87.512,Z 376.627,A -85,B 0,C 180,E1 -28656.346,E2 -28656.346} C_VEL
LIN {X 0,Y 88.362,Z 377.903,A -85,B 0,C 180,E1 -28658.273,E2 -28658.273} C_VEL
LIN {X 0,Y 90.686,Z 381.808,A -85,B 0,C 180,E1 -28662.831,E2 -28662.831} C_VEL
LIN {X 0,Y 93.636,Z 387.018,A -85,B 0,C 180,E1 -28667.568,E2 -28667.568} C_VEL
LIN {X 0,Y 97.804,Z 395.479,A -85,B 0,C 180,E1 -28673.066,E2 -28673.066} C_VEL
LIN {X 0,Y 102.123,Z 405.482,A -85,B 0,C 180,E1 -28677.902,E2 -28677.902} C_VEL
LIN {X 0,Y 98.845,Z 433.767,A -85,B 0,C 180,E1 -28679.4,E2 -28679.4} C_VEL
LIN {X 0,Y 96.22,Z 447.142,A -85,B 0,C 180,E1 -28680.656,E2 -28680.656} C_VEL
LIN {X 0,Y 92.792,Z 459.298,A -85,B 0,C 180,E1 -28682.346,E2 -28682.346} C_VEL
LIN {X 0,Y 88.41,Z 471.112,A -85,B 0,C 180,E1 -28684.691,E2 -28684.691} C_VEL
LIN {X 0,Y 83.013,Z 482.881,A -85,B 0,C 180,E1 -28687.984,E2 -28687.984} C_VEL
LIN {X 0,Y 77.412,Z 493.305,A -85,B 0,C 180,E1 -28692.141,E2 -28692.141} C_VEL
LIN {X 0,Y 71.616,Z 502.838,A -85,B 0,C 180,E1 -28697.592,E2 -28697.592} C_VEL
LIN {X 0,Y 65.488,Z 512.208,A -85,B 0,C 180,E1 -28705.364,E2 -28705.364} C_VEL
LIN {X 0,Y 61.192,Z 518.792,A -85,B 0,C 180,E1 -28713.27,E2 -28713.27} C_VEL
LIN {X 0,Y 57.461,Z 525.149,A -85,B 0,C 180,E1 -28724.135,E2 -28724.135} C_VEL
LIN {X 0,Y 55.832,Z 528.654,A -85,B 0,C 180,E1 -28732.16,E2 -28732.16} C_VEL
LIN {X 0,Y 55.101,Z 532.747,A -85,B 0,C 180,E1 -28744.995,E2 -28744.995} C_VEL
LIN {X 0,Y 56.95,Z 535.53,A -85,B 0,C 180,E1 -28757.731,E2 -28757.731} C_VEL
LIN {X 0,Y 59.538,Z 536.719,A -85,B 0,C 180,E1 -28765.676,E2 -28765.676} C_VEL
LIN {X 0,Y 63.59,Z 537.364,A -85,B 0,C 180,E1 -28773.763,E2 -28773.763} C_VEL
LIN {X 0,Y 70.196,Z 537.211,A -85,B 0,C 180,E1 -28782.521,E2 -28782.521} C_VEL
LIN {X 0,Y 78.49,Z 535.87,A -85,B 0,C 180,E1 -28789.926,E2 -28789.926} C_VEL
LIN {X 0,Y 87.019,Z 533.553,A -85,B 0,C 180,E1 -28795.367,E2 -28795.367} C_VEL
LIN {X 0,Y 96.651,Z 529.951,A -85,B 0,C 180,E1 -28800,E2 -28800} C_VEL
LIN {X 0,Y 106.815,Z 524.974,A -85,B 0,C 180,E1 -28803.772,E2 -28803.772} C_VEL
LIN {X 0,Y 117.395,Z 518.448,A -85,B 0,C 180,E1 -28806.877,E2 -28806.877} C_VEL
LIN {X 0,Y 126.278,Z 511.803,A -85,B 0,C 180,E1 -28809.023,E2 -28809.023} C_VEL
LIN {X 0,Y 135.983,Z 503.053,A -85,B 0,C 180,E1 -28810.966,E2 -28810.966} C_VEL
LIN {X 0,Y 144.839,Z 493.201,A -85,B 0,C 180,E1 -28812.501,E2 -28812.501} C_VEL
LIN {X 0,Y 152.779,Z 482.373,A -85,B 0,C 180,E1 -28813.698,E2 -28813.698} C_VEL
LIN {X 0,Y 158.796,Z 472.239,A -85,B 0,C 180,E1 -28814.55,E2 -28814.55} C_VEL
LIN {X 0,Y 164.546,Z 459.903,A -85,B 0,C 180,E1 -28815.329,E2 -28815.329} C_VEL
LIN {X 0,Y 164.936,Z 458.924,A -85,B 0,C 180,E1 -28815.381,E2 -28815.381} C_VEL
LIN {X 0,Y 164.355,Z 460.458,A -85,B 0,C 180,E1 -28816.025,E2 -28816.025} C_VEL
LIN {X 0,Y 158.548,Z 472.84,A -85,B 0,C 180,E1 -28816.592,E2 -28816.592} C_VEL
LIN {X 0,Y 151.815,Z 484.047,A -85,B 0,C 180,E1 -28817.335,E2 -28817.335} C_VEL
LIN {X 0,Y 144.285,Z 494.252,A -85,B 0,C 180,E1 -28818.268,E2 -28818.268} C_VEL
LIN {X 0,Y 136.067,Z 503.492,A -85,B 0,C 180,E1 -28819.542,E2 -28819.542} C_VEL
LIN {X 0,Y 126.32,Z 512.518,A -85,B 0,C 180,E1 -28821.304,E2 -28821.304} C_VEL
LIN {X 0,Y 115.154,Z 520.962,A -85,B 0,C 180,E1 -28823.764,E2 -28823.764} C_VEL
LIN {X 0,Y 105.914,Z 526.729,A -85,B 0,C 180,E1 -28826.424,E2 -28826.424} C_VEL
LIN {X 0,Y 96.886,Z 531.358,A -85,B 0,C 180,E1 -28829.521,E2 -28829.521} C_VEL
LIN {X 0,Y 88.352,Z 534.949,A -85,B 0,C 180,E1 -28833.394,E2 -28833.394} C_VEL
LIN {X 0,Y 80.333,Z 537.619,A -85,B 0,C 180,E1 -28838.091,E2 -28838.091} C_VEL
LIN {X 0,Y 70.694,Z 539.874,A -85,B 0,C 180,E1 -28845.931,E2 -28845.931} C_VEL
LIN {X 0,Y 62.899,Z 540.612,A -85,B 0,C 180,E1 -28856.064,E2 -28856.064} C_VEL
LIN {X 0,Y 57.818,Z 539.91,A -85,B 0,C 180,E1 -28868.639,E2 -28868.639} C_VEL
LIN {X 0,Y 55.772,Z 537.734,A -85,B 0,C 180,E1 -28882.785,E2 -28882.785} C_VEL
LIN {X 0,Y 55.82,Z 535.998,A -85,B 0,C 180,E1 -28890.023,E2 -28890.023} C_VEL
LIN {X 0,Y 56.062,Z 532.44,A -85,B 0,C 180,E1 -28900.862,E2 -28900.862} C_VEL
LIN {X 0,Y 57.837,Z 527.704,A -85,B 0,C 180,E1 -28911.402,E2 -28911.402} C_VEL
LIN {X 0,Y 62.069,Z 520.552,A -85,B 0,C 180,E1 -28922.559,E2 -28922.559} C_VEL
LIN {X 0,Y 67.239,Z 512.709,A -85,B 0,C 180,E1 -28930.811,E2 -28930.811} C_VEL
LIN {X 0,Y 73.484,Z 503.025,A -85,B 0,C 180,E1 -28937.696,E2 -28937.696} C_VEL
LIN {X 0,Y 79.562,Z 492.678,A -85,B 0,C 180,E1 -28942.678,E2 -28942.678} C_VEL
LIN {X 0,Y 85.396,Z 481.171,A -85,B 0,C 180,E1 -28946.459,E2 -28946.459} C_VEL
LIN {X 0,Y 90.156,Z 469.903,A -85,B 0,C 180,E1 -28949.057,E2 -28949.057} C_VEL
LIN {X 0,Y 94.399,Z 457.252,A -85,B 0,C 180,E1 -28951.041,E2 -28951.041} C_VEL
LIN {X 0,Y 97.724,Z 443.613,A -85,B 0,C 180,E1 -28952.459,E2 -28952.459} C_VEL
LIN {X 0,Y 99.567,Z 431.35,A -85,B 0,C 180,E1 -28953.276,E2 -28953.276} C_VEL
LIN {X 0,Y 101.896,Z 410.109,A -85,B 0,C 180,E1 -28954.348,E2 -28954.348} C_VEL
LIN {X 0,Y 99.07,Z 399.597,A -85,B 0,C 180,E1 -28957.907,E2 -28957.907} C_VEL
LIN {X 0,Y 97.621,Z 395.323,A -85,B 0,C 180,E1 -28959.782,E2 -28959.782} C_VEL
LIN {X 0,Y 93.788,Z 387.231,A -85,B 0,C 180,E1 -28964.908,E2 -28964.908} C_VEL
LIN {X 0,Y 90.084,Z 380.402,A -85,B 0,C 180,E1 -28971.023,E2 -28971.023} C_VEL
LIN {X 0,Y 87.765,Z 376.272,A -85,B 0,C 180,E1 -28975.956,E2 -28975.956} C_VEL
LIN {X 0,Y 85.988,Z 372.881,A -85,B 0,C 180,E1 -28981.061,E2 -28981.061} C_VEL
LIN {X 0,Y 85.645,Z 372.124,A -85,B 0,C 180,E1 -28982.352,E2 -28982.352} C_VEL
LIN {X 0,Y 83.743,Z 370.333,A -85,B 0,C 180,E1 -28992.299,E2 -28992.299} C_VEL
LIN {X 0,Y 83.591,Z 370.573,A -85,B 0,C 180,E1 -28998.44,E2 -28998.44} C_VEL
LIN {X 0,Y 84.794,Z 372.426,A -85,B 0,C 180,E1 -29007.68,E2 -29007.68} C_VEL
LIN {X 0,Y 85.423,Z 373.464,A -85,B 0,C 180,E1 -29010.169,E2 -29010.169} C_VEL
LIN {X 0,Y 86.009,Z 375.281,A -85,B 0,C 180,E1 -29012.45,E2 -29012.45} C_VEL
LIN {X 0,Y 87.096,Z 380.292,A -85,B 0,C 180,E1 -29016.473,E2 -29016.473} C_VEL
LIN {X 0,Y 89.144,Z 388.823,A -85,B 0,C 180,E1 -29022.164,E2 -29022.164} C_VEL
LIN {X 0,Y 90.212,Z 391.198,A -85,B 0,C 180,E1 -29024.194,E2 -29024.194} C_VEL
LIN {X 0,Y 93.716,Z 398.608,A -85,B 0,C 180,E1 -29029.673,E2 -29029.673} C_VEL
LIN {X 0,Y 97.549,Z 408.023,A -85,B 0,C 180,E1 -29034.7,E2 -29034.7} C_VEL
LIN {X 0,Y 96.631,Z 416.884,A -85,B 0,C 180,E1 -29035.212,E2 -29035.212} C_VEL
LIN {X 0,Y 94.076,Z 436.117,A -85,B 0,C 180,E1 -29036.233,E2 -29036.233} C_VEL
LIN {X 0,Y 91.414,Z 448.531,A -85,B 0,C 180,E1 -29037.427,E2 -29037.427} C_VEL
LIN {X 0,Y 87.591,Z 461.055,A -85,B 0,C 180,E1 -29039.221,E2 -29039.221} C_VEL
LIN {X 0,Y 82.98,Z 472.576,A -85,B 0,C 180,E1 -29041.533,E2 -29041.533} C_VEL
LIN {X 0,Y 77.241,Z 484.28,A -85,B 0,C 180,E1 -29044.889,E2 -29044.889} C_VEL
LIN {X 0,Y 70.758,Z 495.385,A -85,B 0,C 180,E1 -29049.639,E2 -29049.639} C_VEL
LIN {X 0,Y 64.602,Z 504.68,A -85,B 0,C 180,E1 -29055.453,E2 -29055.453} C_VEL
LIN {X 0,Y 58.71,Z 512.959,A -85,B 0,C 180,E1 -29063.103,E2 -29063.103} C_VEL
LIN {X 0,Y 53.278,Z 520.588,A -85,B 0,C 180,E1 -29073.757,E2 -29073.757} C_VEL
LIN {X 0,Y 49.665,Z 526.657,A -85,B 0,C 180,E1 -29086.412,E2 -29086.412} C_VEL
LIN {X 0,Y 48.042,Z 530.757,A -85,B 0,C 180,E1 -29098.629,E2 -29098.629} C_VEL
LIN {X 0,Y 48.946,Z 534.454,A -85,B 0,C 180,E1 -29114.116,E2 -29114.116} C_VEL
LIN {X 0,Y 52.715,Z 536.672,A -85,B 0,C 180,E1 -29127.772,E2 -29127.772} C_VEL
LIN {X 0,Y 59.66,Z 537.713,A -85,B 0,C 180,E1 -29140.383,E2 -29140.383} C_VEL
LIN {X 0,Y 66.177,Z 537.498,A -85,B 0,C 180,E1 -29147.737,E2 -29147.737} C_VEL
LIN {X 0,Y 74.873,Z 536.246,A -85,B 0,C 180,E1 -29154.614,E2 -29154.614} C_VEL
LIN {X 0,Y 84.485,Z 533.848,A -85,B 0,C 180,E1 -29160,E2 -29160} C_VEL
LIN {X 0,Y 94.678,Z 530.242,A -85,B 0,C 180,E1 -29164.257,E2 -29164.257} C_VEL
LIN {X 0,Y 106.416,Z 524.688,A -85,B 0,C 180,E1 -29167.963,E2 -29167.963} C_VEL
LIN {X 0,Y 116.357,Z 518.751,A -85,B 0,C 180,E1 -29170.44,E2 -29170.44} C_VEL
LIN {X 0,Y 125.501,Z 512.113,A -85,B 0,C 180,E1 -29172.32,E2 -29172.32} C_VEL
LIN {X 0,Y 135.811,Z 502.993,A -85,B 0,C 180,E1 -29174.058,E2 -29174.058} C_VEL
LIN {X 0,Y 142.093,Z 496.324,A -85,B 0,C 180,E1 -29174.992,E2 -29174.992} C_VEL
LIN {X 0,Y 140.693,Z 497.947,A -85,B 0,C 180,E1 -29175.799,E2 -29175.799} C_VEL
LIN {X 0,Y 132.228,Z 506.598,A -85,B 0,C 180,E1 -29176.967,E2 -29176.967} C_VEL
LIN {X 0,Y 122.299,Z 515.017,A -85,B 0,C 180,E1 -29178.571,E2 -29178.571} C_VEL
LIN {X 0,Y 112.505,Z 521.829,A -85,B 0,C 180,E1 -29180.486,E2 -29180.486} C_VEL
LIN {X 0,Y 102.965,Z 527.343,A -85,B 0,C 180,E1 -29182.902,E2 -29182.902} C_VEL
LIN {X 0,Y 93.604,Z 531.782,A -85,B 0,C 180,E1 -29185.753,E2 -29185.753} C_VEL
LIN {X 0,Y 81.765,Z 536.133,A -85,B 0,C 180,E1 -29190.774,E2 -29190.774} C_VEL
LIN {X 0,Y 70.815,Z 538.937,A -85,B 0,C 180,E1 -29197.479,E2 -29197.479} C_VEL
LIN {X 0,Y 61.214,Z 540.207,A -85,B 0,C 180,E1 -29206.493,E2 -29206.493} C_VEL
LIN {X 0,Y 53.803,Z 540.057,A -85,B 0,C 180,E1 -29218.531,E2 -29218.531} C_VEL
LIN {X 0,Y 49.55,Z 538.448,A -85,B 0,C 180,E1 -29233.549,E2 -29233.549} C_VEL
LIN {X 0,Y 48.746,Z 537.051,A -85,B 0,C 180,E1 -29241.738,E2 -29241.738} C_VEL
LIN {X 0,Y 48.747,Z 535.246,A -85,B 0,C 180,E1 -29250.027,E2 -29250.027} C_VEL
LIN {X 0,Y 49.105,Z 531.533,A -85,B 0,C 180,E1 -29262.423,E2 -29262.423} C_VEL
LIN {X 0,Y 51.278,Z 526.631,A -85,B 0,C 180,E1 -29274.305,E2 -29274.305} C_VEL
LIN {X 0,Y 55.349,Z 520.414,A -85,B 0,C 180,E1 -29284.873,E2 -29284.873} C_VEL
LIN {X 0,Y 60.971,Z 512.62,A -85,B 0,C 180,E1 -29293.783,E2 -29293.783} C_VEL
LIN {X 0,Y 67.125,Z 503.801,A -85,B 0,C 180,E1 -29300.481,E2 -29300.481} C_VEL
LIN {X 0,Y 73.452,Z 493.788,A -85,B 0,C 180,E1 -29305.64,E2 -29305.64} C_VEL
LIN {X 0,Y 79.565,Z 482.649,A -85,B 0,C 180,E1 -29309.48,E2 -29309.48} C_VEL
LIN {X 0,Y 84.528,Z 471.782,A -85,B 0,C 180,E1 -29312.081,E2 -29312.081} C_VEL
LIN {X 0,Y 88.94,Z 459.928,A -85,B 0,C 180,E1 -29314.032,E2 -29314.032} C_VEL
LIN {X 0,Y 92.488,Z 447.145,A -85,B 0,C 180,E1 -29315.46,E2 -29315.46} C_VEL
LIN {X 0,Y 94.949,Z 433.325,A -85,B 0,C 180,E1 -29316.442,E2 -29316.442} C_VEL
LIN {X 0,Y 97.402,Z 411.895,A -85,B 0,C 180,E1 -29317.531,E2 -29317.531} C_VEL
LIN {X 0,Y 94.989,Z 402.17,A -85,B 0,C 180,E1 -29321.174,E2 -29321.174} C_VEL
LIN {X 0,Y 92.855,Z 396.792,A -85,B 0,C 180,E1 -29324.233,E2 -29324.233} C_VEL
LIN {X 0,Y 90.192,Z 391.157,A -85,B 0,C 180,E1 -29328.504,E2 -29328.504} C_VEL
LIN {X 0,Y 87.844,Z 386.365,A -85,B 0,C 180,E1 -29333.138,E2 -29333.138} C_VEL
LIN {X 0,Y 85.804,Z 382.431,A -85,B 0,C 180,E1 -29338.092,E2 -29338.092} C_VEL
LIN {X 0,Y 84.265,Z 378.98,A -85,B 0,C 180,E1 -29343.586,E2 -29343.586} C_VEL
LIN {X 0,Y 82.73,Z 377.366,A -85,B 0,C 180,E1 -29352.452,E2 -29352.452} C_VEL
LIN {X 0,Y 82.596,Z 377.66,A -85,B 0,C 180,E1 -29358.67,E2 -29358.67} C_VEL
LIN {X 0,Y 84.291,Z 380.022,A -85,B 0,C 180,E1 -29369.627,E2 -29369.627} C_VEL
LIN {X 0,Y 86.047,Z 383.414,A -85,B 0,C 180,E1 -29375.42,E2 -29375.42} C_VEL
LIN {X 0,Y 88.606,Z 388.121,A -85,B 0,C 180,E1 -29381.187,E2 -29381.187} C_VEL
LIN {X 0,Y 90.212,Z 391.198,A -85,B 0,C 180,E1 -29384.194,E2 -29384.194} C_VEL
LIN {X 0,Y 91.119,Z 393.862,A -85,B 0,C 180,E1 -29385.898,E2 -29385.898} C_VEL
LIN {X 0,Y 91.598,Z 397.291,A -85,B 0,C 180,E1 -29387.127,E2 -29387.127} C_VEL
LIN {X 0,Y 92.39,Z 407.351,A -85,B 0,C 180,E1 -29389.789,E2 -29389.789} C_VEL
LIN {X 0,Y 92.922,Z 409.589,A -85,B 0,C 180,E1 -29390.705,E2 -29390.705} C_VEL
LIN {X 0,Y 93.338,Z 410.735,A -85,B 0,C 180,E1 -29391.3,E2 -29391.3} C_VEL
LIN {X 0,Y 90.44,Z 433.881,A -85,B 0,C 180,E1 -29392.474,E2 -29392.474} C_VEL
LIN {X 0,Y 87.431,Z 447.911,A -85,B 0,C 180,E1 -29393.689,E2 -29393.689} C_VEL
LIN {X 0,Y 83.48,Z 460.541,A -85,B 0,C 180,E1 -29395.354,E2 -29395.354} C_VEL
LIN {X 0,Y 78.639,Z 472.198,A -85,B 0,C 180,E1 -29397.556,E2 -29397.556} C_VEL
LIN {X 0,Y 72.368,Z 484.403,A -85,B 0,C 180,E1 -29400.931,E2 -29400.931} C_VEL
LIN {X 0,Y 65.695,Z 495.207,A -85,B 0,C 180,E1 -29405.489,E2 -29405.489} C_VEL
LIN {X 0,Y 58.919,Z 504.735,A -85,B 0,C 180,E1 -29411.497,E2 -29411.497} C_VEL
LIN {X 0,Y 53.174,Z 512.187,A -85,B 0,C 180,E1 -29418.541,E2 -29418.541} C_VEL
LIN {X 0,Y 47.002,Z 520.054,A -85,B 0,C 180,E1 -29429.972,E2 -29429.972} C_VEL
LIN {X 0,Y 43.182,Z 525.633,A -85,B 0,C 180,E1 -29442.438,E2 -29442.438} C_VEL
LIN {X 0,Y 41.18,Z 529.667,A -85,B 0,C 180,E1 -29455.098,E2 -29455.098} C_VEL
LIN {X 0,Y 41.498,Z 533.659,A -85,B 0,C 180,E1 -29472.597,E2 -29472.597} C_VEL
LIN {X 0,Y 43.674,Z 535.591,A -85,B 0,C 180,E1 -29483.515,E2 -29483.515} C_VEL
LIN {X 0,Y 47.281,Z 536.958,A -85,B 0,C 180,E1 -29493.517,E2 -29493.517} C_VEL
LIN {X 0,Y 54.233,Z 537.935,A -85,B 0,C 180,E1 -29504.978,E2 -29504.978} C_VEL
LIN {X 0,Y 63.548,Z 537.734,A -85,B 0,C 180,E1 -29514.22,E2 -29514.22} C_VEL
LIN {X 0,Y 72.233,Z 536.547,A -85,B 0,C 180,E1 -29520,E2 -29520} C_VEL
LIN {X 0,Y 82.521,Z 534.159,A -85,B 0,C 180,E1 -29524.885,E2 -29524.885} C_VEL
LIN {X 0,Y 93.287,Z 530.564,A -85,B 0,C 180,E1 -29528.666,E2 -29528.666} C_VEL
LIN {X 0,Y 104.433,Z 525.572,A -85,B 0,C 180,E1 -29531.647,E2 -29531.647} C_VEL
LIN {X 0,Y 115.886,Z 518.988,A -85,B 0,C 180,E1 -29534.054,E2 -29534.054} C_VEL
LIN {X 0,Y 120.698,Z 515.73,A -85,B 0,C 180,E1 -29534.91,E2 -29534.91} C_VEL
LIN {X 0,Y 118.235,Z 517.534,A -85,B 0,C 180,E1 -29535.705,E2 -29535.705} C_VEL
LIN {X 0,Y 110.242,Z 522.654,A -85,B 0,C 180,E1 -29537.062,E2 -29537.062} C_VEL
LIN {X 0,Y 100.424,Z 527.956,A -85,B 0,C 180,E1 -29539.181,E2 -29539.181} C_VEL
LIN {X 0,Y 90.749,Z 532.183,A -85,B 0,C 180,E1 -29541.717,E2 -29541.717} C_VEL
LIN {X 0,Y 78.367,Z 536.325,A -85,B 0,C 180,E1 -29546.305,E2 -29546.305} C_VEL
LIN {X 0,Y 66.724,Z 538.881,A -85,B 0,C 180,E1 -29552.624,E2 -29552.624} C_VEL
LIN {X 0,Y 56.272,Z 539.982,A -85,B 0,C 180,E1 -29561.504,E2 -29561.504} C_VEL
LIN {X 0,Y 47.863,Z 539.655,A -85,B 0,C 180,E1 -29574.068,E2 -29574.068} C_VEL
LIN {X 0,Y 42.794,Z 537.835,A -85,B 0,C 180,E1 -29590.859,E2 -29590.859} C_VEL
LIN {X 0,Y 41.755,Z 536.36,A -85,B 0,C 180,E1 -29600.343,E2 -29600.343} C_VEL
LIN {X 0,Y 41.668,Z 534.472,A -85,B 0,C 180,E1 -29610.031,E2 -29610.031} C_VEL
LIN {X 0,Y 42.207,Z 530.586,A -85,B 0,C 180,E1 -29624.495,E2 -29624.495} C_VEL
LIN {X 0,Y 45.559,Z 524.5,A -85,B 0,C 180,E1 -29640.12,E2 -29640.12} C_VEL
LIN {X 0,Y 50.645,Z 517.806,A -85,B 0,C 180,E1 -29651.267,E2 -29651.267} C_VEL
LIN {X 0,Y 57.18,Z 509.455,A -85,B 0,C 180,E1 -29660.222,E2 -29660.222} C_VEL
LIN {X 0,Y 63.553,Z 500.813,A -85,B 0,C 180,E1 -29666.148,E2 -29666.148} C_VEL
LIN {X 0,Y 70.383,Z 490.278,A -85,B 0,C 180,E1 -29670.926,E2 -29670.926} C_VEL
LIN {X 0,Y 76.205,Z 479.837,A -85,B 0,C 180,E1 -29674.083,E2 -29674.083} C_VEL
LIN {X 0,Y 81.442,Z 468.336,A -85,B 0,C 180,E1 -29676.505,E2 -29676.505} C_VEL
LIN {X 0,Y 86.064,Z 455.349,A -85,B 0,C 180,E1 -29678.293,E2 -29678.293} C_VEL
LIN {X 0,Y 89.443,Z 442.058,A -85,B 0,C 180,E1 -29679.507,E2 -29679.507} C_VEL
LIN {X 0,Y 91.652,Z 427.368,A -85,B 0,C 180,E1 -29680.326,E2 -29680.326} C_VEL
LIN {X 0,Y 93.255,Z 413.904,A -85,B 0,C 180,E1 -29680.96,E2 -29680.96} C_VEL
LIN {X 0,Y 91.253,Z 405.386,A -85,B 0,C 180,E1 -29684.457,E2 -29684.457} C_VEL
LIN {X 0,Y 88.378,Z 398.267,A -85,B 0,C 180,E1 -29689.478,E2 -29689.478} C_VEL
LIN {X 0,Y 85.946,Z 392.764,A -85,B 0,C 180,E1 -29694.733,E2 -29694.733} C_VEL
LIN {X 0,Y 84.069,Z 388.759,A -85,B 0,C 180,E1 -29700,E2 -29700} C_VEL
LIN {X 0,Y 82.917,Z 385.818,A -85,B 0,C 180,E1 -29704.862,E2 -29704.862} C_VEL
LIN {X 0,Y 81.717,Z 384.404,A -85,B 0,C 180,E1 -29712.609,E2 -29712.609} C_VEL
LIN {X 0,Y 81.594,Z 384.708,A -85,B 0,C 180,E1 -29718.615,E2 -29718.615} C_VEL
LIN {X 0,Y 82.906,Z 386.827,A -85,B 0,C 180,E1 -29728.347,E2 -29728.347} C_VEL
LIN {X 0,Y 84.791,Z 390.823,A -85,B 0,C 180,E1 -29735.084,E2 -29735.084} C_VEL
LIN {X 0,Y 86.712,Z 394.784,A -85,B 0,C 180,E1 -29739.817,E2 -29739.817} C_VEL
LIN {X 0,Y 88.636,Z 398.923,A -85,B 0,C 180,E1 -29743.689,E2 -29743.689} C_VEL
LIN {X 0,Y 91.571,Z 406.024,A -85,B 0,C 180,E1 -29748.689,E2 -29748.689} C_VEL
LIN {X 0,Y 92.922,Z 409.589,A -85,B 0,C 180,E1 -29750.705,E2 -29750.705} C_VEL
LIN {X 0,Y 93.129,Z 411.786,A -85,B 0,C 180,E1 -29751.263,E2 -29751.263} C_VEL
LIN {X 0,Y 92.617,Z 414.871,A -85,B 0,C 180,E1 -29751.251,E2 -29751.251} C_VEL
LIN {X 0,Y 91.134,Z 419.102,A -85,B 0,C 180,E1 -29750.454,E2 -29750.454} C_VEL
LIN {X 0,Y 88.43,Z 425.593,A -85,B 0,C 180,E1 -29748.714,E2 -29748.714} C_VEL
LIN {X 0,Y 87.487,Z 429.098,A -85,B 0,C 180,E1 -29748.354,E2 -29748.354} C_VEL
LIN {X 0,Y 87.367,Z 429.822,A -85,B 0,C 180,E1 -29748.374,E2 -29748.374} C_VEL
LIN {X 0,Y 84.661,Z 443.909,A -85,B 0,C 180,E1 -29749.29,E2 -29749.29} C_VEL
LIN {X 0,Y 81.206,Z 455.806,A -85,B 0,C 180,E1 -29750.558,E2 -29750.558} C_VEL
LIN {X 0,Y 76.419,Z 468.062,A -85,B 0,C 180,E1 -29752.444,E2 -29752.444} C_VEL
LIN {X 0,Y 70.714,Z 479.549,A -85,B 0,C 180,E1 -29754.978,E2 -29754.978} C_VEL
LIN {X 0,Y 64.142,Z 490.444,A -85,B 0,C 180,E1 -29758.616,E2 -29758.616} C_VEL
LIN {X 0,Y 56.463,Z 501.168,A -85,B 0,C 180,E1 -29764.15,E2 -29764.15} C_VEL
LIN {X 0,Y 49.353,Z 509.88,A -85,B 0,C 180,E1 -29771.286,E2 -29771.286} C_VEL
LIN {X 0,Y 42.626,Z 517.591,A -85,B 0,C 180,E1 -29781.594,E2 -29781.594} C_VEL
LIN {X 0,Y 37.407,Z 523.923,A -85,B 0,C 180,E1 -29795.355,E2 -29795.355} C_VEL
LIN {X 0,Y 34.906,Z 527.736,A -85,B 0,C 180,E1 -29807.532,E2 -29807.532} C_VEL
LIN {X 0,Y 33.97,Z 532.302,A -85,B 0,C 180,E1 -29828.312,E2 -29828.312} C_VEL
LIN {X 0,Y 36.377,Z 535.047,A -85,B 0,C 180,E1 -29844.577,E2 -29844.577} C_VEL
LIN {X 0,Y 42.401,Z 537.233,A -85,B 0,C 180,E1 -29860.64,E2 -29860.64} C_VEL
LIN {X 0,Y 50.518,Z 538.219,A -85,B 0,C 180,E1 -29872.003,E2 -29872.003} C_VEL
LIN {X 0,Y 60.004,Z 538.091,A -85,B 0,C 180,E1 -29880,E2 -29880} C_VEL
LIN {X 0,Y 70.623,Z 536.81,A -85,B 0,C 180,E1 -29885.877,E2 -29885.877} C_VEL
LIN {X 0,Y 81.173,Z 534.493,A -85,B 0,C 180,E1 -29889.972,E2 -29889.972} C_VEL
LIN {X 0,Y 93.942,Z 530.314,A -85,B 0,C 180,E1 -29893.53,E2 -29893.53} C_VEL
LIN {X 0,Y 98.96,Z 528.239,A -85,B 0,C 180,E1 -29894.659,E2 -29894.659} C_VEL
LIN {X 0,Y 96.392,Z 529.408,A -85,B 0,C 180,E1 -29895.667,E2 -29895.667} C_VEL
LIN {X 0,Y 85.102,Z 533.704,A -85,B 0,C 180,E1 -29898.311,E2 -29898.311} C_VEL
LIN {X 0,Y 75.483,Z 536.474,A -85,B 0,C 180,E1 -29901.455,E2 -29901.455} C_VEL
LIN {X 0,Y 63.174,Z 538.825,A -85,B 0,C 180,E1 -29907.181,E2 -29907.181} C_VEL
LIN {X 0,Y 51.827,Z 539.747,A -85,B 0,C 180,E1 -29915.597,E2 -29915.597} C_VEL
LIN {X 0,Y 42.301,Z 539.183,A -85,B 0,C 180,E1 -29928.395,E2 -29928.395} C_VEL
LIN {X 0,Y 36.174,Z 537.21,A -85,B 0,C 180,E1 -29947.176,E2 -29947.176} C_VEL
LIN {X 0,Y 34.545,Z 534.691,A -85,B 0,C 180,E1 -29964.2,E2 -29964.2} C_VEL
LIN {X 0,Y 34.607,Z 533.643,A -85,B 0,C 180,E1 -29970.038,E2 -29970.038} C_VEL
LIN {X 0,Y 35.364,Z 529.579,A -85,B 0,C 180,E1 -29987.381,E2 -29987.381} C_VEL
LIN {X 0,Y 39.575,Z 523.27,A -85,B 0,C 180,E1 -30005.288,E2 -30005.288} C_VEL
LIN {X 0,Y 45.539,Z 516.361,A -85,B 0,C 180,E1 -30017.182,E2 -30017.182} C_VEL
LIN {X 0,Y 51.602,Z 509.266,A -85,B 0,C 180,E1 -30024.842,E2 -30024.842} C_VEL
LIN {X 0,Y 59.248,Z 499.556,A -85,B 0,C 180,E1 -30031.361,E2 -30031.361} C_VEL
LIN {X 0,Y 66.467,Z 488.962,A -85,B 0,C 180,E1 -30035.82,E2 -30035.82} C_VEL
LIN {X 0,Y 72.613,Z 478.275,A -85,B 0,C 180,E1 -30038.721,E2 -30038.721} C_VEL
LIN {X 0,Y 78.091,Z 466.321,A -85,B 0,C 180,E1 -30040.944,E2 -30040.944} C_VEL
LIN {X 0,Y 82.428,Z 454.273,A -85,B 0,C 180,E1 -30042.409,E2 -30042.409} C_VEL
LIN {X 0,Y 85.731,Z 441.439,A -85,B 0,C 180,E1 -30043.461,E2 -30043.461} C_VEL
LIN {X 0,Y 87.902,Z 427.508,A -85,B 0,C 180,E1 -30044.179,E2 -30044.179} C_VEL
LIN {X 0,Y 89.328,Z 415.794,A -85,B 0,C 180,E1 -30044.724,E2 -30044.724} C_VEL
LIN {X 0,Y 88.013,Z 409.601,A -85,B 0,C 180,E1 -30047.549,E2 -30047.549} C_VEL
LIN {X 0,Y 85.856,Z 403.61,A -85,B 0,C 180,E1 -30052.09,E2 -30052.09} C_VEL
LIN {X 0,Y 83.774,Z 398.466,A -85,B 0,C 180,E1 -30057.333,E2 -30057.333} C_VEL
LIN {X 0,Y 82.416,Z 395.029,A -85,B 0,C 180,E1 -30062.056,E2 -30062.056} C_VEL
LIN {X 0,Y 81.62,Z 392.657,A -85,B 0,C 180,E1 -30066.037,E2 -30066.037} C_VEL
LIN {X 0,Y 80.705,Z 391.441,A -85,B 0,C 180,E1 -30072.77,E2 -30072.77} C_VEL
LIN {X 0,Y 80.594,Z 391.836,A -85,B 0,C 180,E1 -30078.855,E2 -30078.855} C_VEL
LIN {X 0,Y 81.602,Z 393.735,A -85,B 0,C 180,E1 -30087.233,E2 -30087.233} C_VEL
LIN {X 0,Y 83.116,Z 397.324,A -85,B 0,C 180,E1 -30093.424,E2 -30093.424} C_VEL
LIN {X 0,Y 84.61,Z 400.802,A -85,B 0,C 180,E1 -30097.728,E2 -30097.728} C_VEL
LIN {X 0,Y 86.405,Z 405.119,A -85,B 0,C 180,E1 -30101.823,E2 -30101.823} C_VEL
LIN {X 0,Y 88.675,Z 411.368,A -85,B 0,C 180,E1 -30106.321,E2 -30106.321} C_VEL
LIN {X 0,Y 89.365,Z 413.425,A -85,B 0,C 180,E1 -30107.552,E2 -30107.552} C_VEL
LIN {X 0,Y 87.367,Z 429.822,A -85,B 0,C 180,E1 -30108.374,E2 -30108.374} C_VEL
LIN {X 0,Y 86.619,Z 433.687,A -85,B 0,C 180,E1 -30108.38,E2 -30108.38} C_VEL
LIN {X 0,Y 84.213,Z 441.166,A -85,B 0,C 180,E1 -30107.759,E2 -30107.759} C_VEL
LIN {X 0,Y 78.751,Z 453.798,A -85,B 0,C 180,E1 -30106.31,E2 -30106.31} C_VEL
LIN {X 0,Y 76.511,Z 459.279,A -85,B 0,C 180,E1 -30106.517,E2 -30106.517} C_VEL
LIN {X 0,Y 71.33,Z 471.24,A -85,B 0,C 180,E1 -30108.292,E2 -30108.292} C_VEL
LIN {X 0,Y 64.935,Z 482.806,A -85,B 0,C 180,E1 -30110.856,E2 -30110.856} C_VEL
LIN {X 0,Y 57.667,Z 493.681,A -85,B 0,C 180,E1 -30114.602,E2 -30114.602} C_VEL
LIN {X 0,Y 49.824,Z 503.478,A -85,B 0,C 180,E1 -30119.985,E2 -30119.985} C_VEL
LIN {X 0,Y 42.041,Z 512.028,A -85,B 0,C 180,E1 -30127.874,E2 -30127.874} C_VEL
LIN {X 0,Y 35.373,Z 518.837,A -85,B 0,C 180,E1 -30138.503,E2 -30138.503} C_VEL
LIN {X 0,Y 29.753,Z 524.983,A -85,B 0,C 180,E1 -30155.093,E2 -30155.093} C_VEL
LIN {X 0,Y 27.076,Z 529.074,A -85,B 0,C 180,E1 -30172.86,E2 -30172.86} C_VEL
LIN {X 0,Y 27.866,Z 533.39,A -85,B 0,C 180,E1 -30199.09,E2 -30199.09} C_VEL
LIN {X 0,Y 31.194,Z 535.505,A -85,B 0,C 180,E1 -30214.213,E2 -30214.213} C_VEL
LIN {X 0,Y 38.32,Z 537.502,A -85,B 0,C 180,E1 -30229.432,E2 -30229.432} C_VEL
LIN {X 0,Y 49.181,Z 538.563,A -85,B 0,C 180,E1 -30241.207,E2 -30241.207} C_VEL
LIN {X 0,Y 58.142,Z 538.391,A -85,B 0,C 180,E1 -30246.942,E2 -30246.942} C_VEL
LIN {X 0,Y 69.16,Z 537.173,A -85,B 0,C 180,E1 -30251.726,E2 -30251.726} C_VEL
LIN {X 0,Y 77.554,Z 535.552,A -85,B 0,C 180,E1 -30254.383,E2 -30254.383} C_VEL
LIN {X 0,Y 74.726,Z 536.258,A -85,B 0,C 180,E1 -30255.81,E2 -30255.81} C_VEL
LIN {X 0,Y 66.648,Z 537.873,A -85,B 0,C 180,E1 -30258.442,E2 -30258.442} C_VEL
LIN {X 0,Y 54.01,Z 539.283,A -85,B 0,C 180,E1 -30264.441,E2 -30264.441} C_VEL
LIN {X 0,Y 42.396,Z 539.251,A -85,B 0,C 180,E1 -30274.08,E2 -30274.08} C_VEL
LIN {X 0,Y 33.003,Z 537.824,A -85,B 0,C 180,E1 -30290.348,E2 -30290.348} C_VEL
LIN {X 0,Y 29.776,Z 536.551,A -85,B 0,C 180,E1 -30301.884,E2 -30301.884} C_VEL
LIN {X 0,Y 27.547,Z 533.885,A -85,B 0,C 180,E1 -30322.719,E2 -30322.719} C_VEL
LIN {X 0,Y 27.525,Z 532.748,A -85,B 0,C 180,E1 -30330.048,E2 -30330.048} C_VEL
LIN {X 0,Y 28.661,Z 528.507,A -85,B 0,C 180,E1 -30351.628,E2 -30351.628} C_VEL
LIN {X 0,Y 33.031,Z 523.023,A -85,B 0,C 180,E1 -30369.714,E2 -30369.714} C_VEL
LIN {X 0,Y 39.752,Z 516.135,A -85,B 0,C 180,E1 -30382.76,E2 -30382.76} C_VEL
LIN {X 0,Y 46.437,Z 509.069,A -85,B 0,C 180,E1 -30390.537,E2 -30390.537} C_VEL
LIN {X 0,Y 54.663,Z 499.391,A -85,B 0,C 180,E1 -30396.8,E2 -30396.8} C_VEL
LIN {X 0,Y 62.293,Z 488.809,A -85,B 0,C 180,E1 -30400.942,E2 -30400.942} C_VEL
LIN {X 0,Y 68.719,Z 478.153,A -85,B 0,C 180,E1 -30403.549,E2 -30403.549} C_VEL
LIN {X 0,Y 74.423,Z 466.248,A -85,B 0,C 180,E1 -30405.508,E2 -30405.508} C_VEL
LIN {X 0,Y 78.975,Z 454.066,A -85,B 0,C 180,E1 -30406.794,E2 -30406.794} C_VEL
LIN {X 0,Y 82.413,Z 441.097,A -85,B 0,C 180,E1 -30407.727,E2 -30407.727} C_VEL
LIN {X 0,Y 84.856,Z 425.667,A -85,B 0,C 180,E1 -30408.406,E2 -30408.406} C_VEL
LIN {X 0,Y 85.824,Z 417.876,A -85,B 0,C 180,E1 -30408.762,E2 -30408.762} C_VEL
LIN {X 0,Y 85.124,Z 414.177,A -85,B 0,C 180,E1 -30410.661,E2 -30410.661} C_VEL
LIN {X 0,Y 83.402,Z 408.856,A -85,B 0,C 180,E1 -30414.95,E2 -30414.95} C_VEL
LIN {X 0,Y 81.886,Z 404.465,A -85,B 0,C 180,E1 -30419.685,E2 -30419.685} C_VEL
LIN {X 0,Y 80.914,Z 401.424,A -85,B 0,C 180,E1 -30423.976,E2 -30423.976} C_VEL
LIN {X 0,Y 80.359,Z 399.489,A -85,B 0,C 180,E1 -30427.249,E2 -30427.249} C_VEL
LIN {X 0,Y 79.641,Z 398.454,A -85,B 0,C 180,E1 -30433.851,E2 -30433.851} C_VEL
LIN {X 0,Y 79.622,Z 399.126,A -85,B 0,C 180,E1 -30439.883,E2 -30439.883} C_VEL
LIN {X 0,Y 80.341,Z 400.612,A -85,B 0,C 180,E1 -30446.116,E2 -30446.116} C_VEL
LIN {X 0,Y 81.57,Z 403.947,A -85,B 0,C 180,E1 -30451.907,E2 -30451.907} C_VEL
LIN {X 0,Y 83.215,Z 408.312,A -85,B 0,C 180,E1 -30457.22,E2 -30457.22} C_VEL
LIN {X 0,Y 85.539,Z 415.29,A -85,B 0,C 180,E1 -30462.886,E2 -30462.886} C_VEL
LIN {X 0,Y 85.834,Z 416.317,A -85,B 0,C 180,E1 -30463.558,E2 -30463.558} C_VEL
LIN {X 0,Y 83.181,Z 435.224,A -85,B 0,C 180,E1 -30464.374,E2 -30464.374} C_VEL
LIN {X 0,Y 80.043,Z 448.621,A -85,B 0,C 180,E1 -30465.359,E2 -30465.359} C_VEL
LIN {X 0,Y 76.511,Z 459.279,A -85,B 0,C 180,E1 -30466.517,E2 -30466.517} C_VEL
LIN {X 0,Y 74.067,Z 464.659,A -85,B 0,C 180,E1 -30466.749,E2 -30466.749} C_VEL
LIN {X 0,Y 68.842,Z 473.055,A -85,B 0,C 180,E1 -30465.992,E2 -30465.992} C_VEL
LIN {X 0,Y 62.987,Z 481.06,A -85,B 0,C 180,E1 -30465.335,E2 -30465.335} C_VEL
LIN {X 0,Y 59.533,Z 485.83,A -85,B 0,C 180,E1 -30465.951,E2 -30465.951} C_VEL
LIN {X 0,Y 51.565,Z 496.589,A -85,B 0,C 180,E1 -30469.624,E2 -30469.624} C_VEL
LIN {X 0,Y 42.83,Z 506.396,A -85,B 0,C 180,E1 -30475.132,E2 -30475.132} C_VEL
LIN {X 0,Y 34.889,Z 514.113,A -85,B 0,C 180,E1 -30483.009,E2 -30483.009} C_VEL
LIN {X 0,Y 26.409,Z 521.737,A -85,B 0,C 180,E1 -30498.437,E2 -30498.437} C_VEL
LIN {X 0,Y 21.347,Z 526.829,A -85,B 0,C 180,E1 -30519.001,E2 -30519.001} C_VEL
LIN {X 0,Y 20.171,Z 532.046,A -85,B 0,C 180,E1 -30555.825,E2 -30555.825} C_VEL
LIN {X 0,Y 26.053,Z 535.572,A -85,B 0,C 180,E1 -30584.35,E2 -30584.35} C_VEL
LIN {X 0,Y 35.329,Z 537.759,A -85,B 0,C 180,E1 -30600,E2 -30600} C_VEL
LIN {X 0,Y 45.917,Z 538.782,A -85,B 0,C 180,E1 -30608.804,E2 -30608.804} C_VEL
LIN {X 0,Y 57.176,Z 538.693,A -85,B 0,C 180,E1 -30614.231,E2 -30614.231} C_VEL
LIN {X 0,Y 51.478,Z 539.062,A -85,B 0,C 180,E1 -30617.222,E2 -30617.222} C_VEL
LIN {X 0,Y 38.865,Z 538.855,A -85,B 0,C 180,E1 -30625.379,E2 -30625.379} C_VEL
LIN {X 0,Y 33.035,Z 538.214,A -85,B 0,C 180,E1 -30631.763,E2 -30631.763} C_VEL
LIN {X 0,Y 23.77,Z 535.829,A -85,B 0,C 180,E1 -30653.819,E2 -30653.819} C_VEL
LIN {X 0,Y 20.581,Z 533.012,A -85,B 0,C 180,E1 -30680.234,E2 -30680.234} C_VEL
LIN {X 0,Y 20.46,Z 531.85,A -85,B 0,C 180,E1 -30690.064,E2 -30690.064} C_VEL
LIN {X 0,Y 22.221,Z 527.417,A -85,B 0,C 180,E1 -30718.387,E2 -30718.387} C_VEL
LIN {X 0,Y 29.139,Z 520.594,A -85,B 0,C 180,E1 -30741.682,E2 -30741.682} C_VEL
LIN {X 0,Y 37.362,Z 513.161,A -85,B 0,C 180,E1 -30753.387,E2 -30753.387} C_VEL
LIN {X 0,Y 44.946,Z 505.543,A -85,B 0,C 180,E1 -30759.824,E2 -30759.824} C_VEL
LIN {X 0,Y 52.517,Z 496.826,A -85,B 0,C 180,E1 -30764.153,E2 -30764.153} C_VEL
LIN {X 0,Y 60.347,Z 486.063,A -85,B 0,C 180,E1 -30767.335,E2 -30767.335} C_VEL
LIN {X 0,Y 67.059,Z 474.797,A -85,B 0,C 180,E1 -30769.357,E2 -30769.357} C_VEL
LIN {X 0,Y 72.554,Z 463.132,A -85,B 0,C 180,E1 -30770.777,E2 -30770.777} C_VEL
LIN {X 0,Y 77.232,Z 449.747,A -85,B 0,C 180,E1 -30771.824,E2 -30771.824} C_VEL
LIN {X 0,Y 80.364,Z 436.741,A -85,B 0,C 180,E1 -30772.463,E2 -30772.463} C_VEL
LIN {X 0,Y 82.71,Z 419.901,A -85,B 0,C 180,E1 -30773.173,E2 -30773.173} C_VEL
LIN {X 0,Y 81.326,Z 414.629,A -85,B 0,C 180,E1 -30777.437,E2 -30777.437} C_VEL
LIN {X 0,Y 80.212,Z 410.649,A -85,B 0,C 180,E1 -30781.848,E2 -30781.848} C_VEL
LIN {X 0,Y 79.408,Z 407.634,A -85,B 0,C 180,E1 -30786.276,E2 -30786.276} C_VEL
LIN {X 0,Y 79.082,Z 406.322,A -85,B 0,C 180,E1 -30788.8,E2 -30788.8} C_VEL
LIN {X 0,Y 78.636,Z 405.48,A -85,B 0,C 180,E1 -30794.032,E2 -30794.032} C_VEL
LIN {X 0,Y 78.63,Z 406.247,A -85,B 0,C 180,E1 -30800.144,E2 -30800.144} C_VEL
LIN {X 0,Y 79.103,Z 407.463,A -85,B 0,C 180,E1 -30804.905,E2 -30804.905} C_VEL
LIN {X 0,Y 80.036,Z 410.427,A -85,B 0,C 180,E1 -30810.128,E2 -30810.128} C_VEL
LIN {X 0,Y 81.382,Z 414.733,A -85,B 0,C 180,E1 -30815.393,E2 -30815.393} C_VEL
LIN {X 0,Y 82.636,Z 419.62,A -85,B 0,C 180,E1 -30819.321,E2 -30819.321} C_VEL
LIN {X 0,Y 79.948,Z 437.082,A -85,B 0,C 180,E1 -30819.938,E2 -30819.938} C_VEL
LIN {X 0,Y 76.623,Z 450.235,A -85,B 0,C 180,E1 -30820.796,E2 -30820.796} C_VEL
LIN {X 0,Y 71.678,Z 463.6,A -85,B 0,C 180,E1 -30822.114,E2 -30822.114} C_VEL
LIN {X 0,Y 65.743,Z 475.683,A -85,B 0,C 180,E1 -30823.79,E2 -30823.79} C_VEL
LIN {X 0,Y 59.533,Z 485.83,A -85,B 0,C 180,E1 -30825.951,E2 -30825.951} C_VEL
LIN {X 0,Y 55.946,Z 490.506,A -85,B 0,C 180,E1 -30826.703,E2 -30826.703} C_VEL
LIN {X 0,Y 49.033,Z 497.585,A -85,B 0,C 180,E1 -30826.446,E2 -30826.446} C_VEL
LIN {X 0,Y 41.661,Z 504.247,A -85,B 0,C 180,E1 -30826.284,E2 -30826.284} C_VEL
LIN {X 0,Y 37.317,Z 508.136,A -85,B 0,C 180,E1 -30827.798,E2 -30827.798} C_VEL
LIN {X 0,Y 28.113,Z 516.052,A -85,B 0,C 180,E1 -30835.719,E2 -30835.719} C_VEL
LIN {X 0,Y 20.072,Z 522.244,A -85,B 0,C 180,E1 -30849.436,E2 -30849.436} C_VEL
LIN {X 0,Y 14.113,Z 527.128,A -85,B 0,C 180,E1 -30875.158,E2 -30875.158} C_VEL
LIN {X 0,Y 14.19,Z 532.31,A -85,B 0,C 180,E1 -30930.31,E2 -30930.31} C_VEL
LIN {X 0,Y 22.83,Z 535.822,A -85,B 0,C 180,E1 -30960,E2 -30960} C_VEL
LIN {X 0,Y 33.745,Z 538.019,A -85,B 0,C 180,E1 -30972.021,E2 -30972.021} C_VEL
LIN {X 0,Y 36.13,Z 538.332,A -85,B 0,C 180,E1 -30973.614,E2 -30973.614} C_VEL
LIN {X 0,Y 36.393,Z 538.404,A -85,B 0,C 180,E1 -30975.229,E2 -30975.229} C_VEL
LIN {X 0,Y 23.852,Z 536.541,A -85,B 0,C 180,E1 -30988.001,E2 -30988.001} C_VEL
LIN {X 0,Y 14.704,Z 533.223,A -85,B 0,C 180,E1 -31021.551,E2 -31021.551} C_VEL
LIN {X 0,Y 13.406,Z 530.877,A -85,B 0,C 180,E1 -31050.098,E2 -31050.098} C_VEL
LIN {X 0,Y 16.339,Z 526.251,A -85,B 0,C 180,E1 -31090.284,E2 -31090.284} C_VEL
LIN {X 0,Y 25.356,Z 519.186,A -85,B 0,C 180,E1 -31114.378,E2 -31114.378} C_VEL
LIN {X 0,Y 34.761,Z 511.474,A -85,B 0,C 180,E1 -31123.936,E2 -31123.936} C_VEL
LIN {X 0,Y 44.7,Z 501.766,A -85,B 0,C 180,E1 -31129.456,E2 -31129.456} C_VEL
LIN {X 0,Y 52.765,Z 492.278,A -85,B 0,C 180,E1 -31132.346,E2 -31132.346} C_VEL
LIN {X 0,Y 60.058,Z 481.824,A -85,B 0,C 180,E1 -31134.257,E2 -31134.257} C_VEL
LIN {X 0,Y 66.113,Z 471.144,A -85,B 0,C 180,E1 -31135.457,E2 -31135.457} C_VEL
LIN {X 0,Y 71.768,Z 458.387,A -85,B 0,C 180,E1 -31136.388,E2 -31136.388} C_VEL
LIN {X 0,Y 75.929,Z 445.422,A -85,B 0,C 180,E1 -31136.994,E2 -31136.994} C_VEL
LIN {X 0,Y 78.721,Z 431.888,A -85,B 0,C 180,E1 -31137.458,E2 -31137.458} C_VEL
LIN {X 0,Y 79.957,Z 422.973,A -85,B 0,C 180,E1 -31137.736,E2 -31137.736} C_VEL
LIN {X 0,Y 78.892,Z 417.9,A -85,B 0,C 180,E1 -31142.707,E2 -31142.707} C_VEL
LIN {X 0,Y 78.072,Z 414.052,A -85,B 0,C 180,E1 -31148.268,E2 -31148.268} C_VEL
LIN {X 0,Y 77.87,Z 413.121,A -85,B 0,C 180,E1 -31150.399,E2 -31150.399} C_VEL
LIN {X 0,Y 77.59,Z 412.568,A -85,B 0,C 180,E1 -31155.768,E2 -31155.768} C_VEL
LIN {X 0,Y 77.882,Z 414.116,A -85,B 0,C 180,E1 -31163.348,E2 -31163.348} C_VEL
LIN {X 0,Y 78.637,Z 417.277,A -85,B 0,C 180,E1 -31168.819,E2 -31168.819} C_VEL
LIN {X 0,Y 79.612,Z 421.321,A -85,B 0,C 180,E1 -31173.487,E2 -31173.487} C_VEL
LIN {X 0,Y 79.906,Z 422.662,A -85,B 0,C 180,E1 -31174.703,E2 -31174.703} C_VEL
LIN {X 0,Y 77.169,Z 439.145,A -85,B 0,C 180,E1 -31175.175,E2 -31175.175} C_VEL
LIN {X 0,Y 73.557,Z 452.128,A -85,B 0,C 180,E1 -31175.845,E2 -31175.845} C_VEL
LIN {X 0,Y 68.618,Z 464.801,A -85,B 0,C 180,E1 -31176.826,E2 -31176.826} C_VEL
LIN {X 0,Y 62.508,Z 476.661,A -85,B 0,C 180,E1 -31178.062,E2 -31178.062} C_VEL
LIN {X 0,Y 55.071,Z 488.064,A -85,B 0,C 180,E1 -31179.998,E2 -31179.998} C_VEL
LIN {X 0,Y 46.813,Z 498.42,A -85,B 0,C 180,E1 -31182.919,E2 -31182.919} C_VEL
LIN {X 0,Y 37.709,Z 507.776,A -85,B 0,C 180,E1 -31187.55,E2 -31187.55} C_VEL
LIN {X 0,Y 37.317,Z 508.136,A -85,B 0,C 180,E1 -31187.798,E2 -31187.798} C_VEL
LIN {X 0,Y 32.856,Z 511.842,A -85,B 0,C 180,E1 -31189.784,E2 -31189.784} C_VEL
LIN {X 0,Y 24.594,Z 517.276,A -85,B 0,C 180,E1 -31191.053,E2 -31191.053} C_VEL
LIN {X 0,Y 15.921,Z 522.153,A -85,B 0,C 180,E1 -31193.525,E2 -31193.525} C_VEL
LIN {X 0,Y 11,Z 524.92,A -85,B 0,C 180,E1 -31201.687,E2 -31201.687} C_VEL
LIN {X 0,Y 5.524,Z 529.611,A -85,B 0,C 180,E1 -31269.192,E2 -31269.192} C_VEL
LIN {X 0,Y 14.276,Z 534.008,A -85,B 0,C 180,E1 -31330.604,E2 -31330.604} C_VEL
LIN {X 0,Y 16.312,Z 534.633,A -85,B 0,C 180,E1 -31333.597,E2 -31333.597} C_VEL
LIN {X 0,Y 14.911,Z 534.296,A -85,B 0,C 180,E1 -31339.766,E2 -31339.766} C_VEL
LIN {X 0,Y 7.12,Z 531.159,A -85,B 0,C 180,E1 -31380.64,E2 -31380.64} C_VEL
LIN {X 0,Y 6.328,Z 529.836,A -85,B 0,C 180,E1 -31410.207,E2 -31410.207} C_VEL
LIN {X 0,Y 11.846,Z 524.996,A -85,B 0,C 180,E1 -31473.102,E2 -31473.102} C_VEL
LIN {X 0,Y 21.498,Z 518.834,A -85,B 0,C 180,E1 -31489.04,E2 -31489.04} C_VEL
LIN {X 0,Y 31.766,Z 511.117,A -85,B 0,C 180,E1 -31495.04,E2 -31495.04} C_VEL
LIN {X 0,Y 42.209,Z 501.42,A -85,B 0,C 180,E1 -31498.206,E2 -31498.206} C_VEL
LIN {X 0,Y 50.966,Z 491.396,A -85,B 0,C 180,E1 -31499.889,E2 -31499.889} C_VEL
LIN {X 0,Y 58.886,Z 480.083,A -85,B 0,C 180,E1 -31500.922,E2 -31500.922} C_VEL
LIN {X 0,Y 65.05,Z 469.087,A -85,B 0,C 180,E1 -31501.519,E2 -31501.519} C_VEL
LIN {X 0,Y 70.339,Z 456.927,A -85,B 0,C 180,E1 -31501.953,E2 -31501.953} C_VEL
LIN {X 0,Y 74.576,Z 443.285,A -85,B 0,C 180,E1 -31502.248,E2 -31502.248} C_VEL
LIN {X 0,Y 77.072,Z 430.729,A -85,B 0,C 180,E1 -31502.533,E2 -31502.533} C_VEL
LIN {X 0,Y 77.673,Z 426.174,A -85,B 0,C 180,E1 -31502.774,E2 -31502.774} C_VEL
LIN {X 0,Y 77.095,Z 422.598,A -85,B 0,C 180,E1 -31507.01,E2 -31507.01} C_VEL
LIN {X 0,Y 76.806,Z 420.1,A -85,B 0,C 180,E1 -31510.978,E2 -31510.978} C_VEL
LIN {X 0,Y 76.582,Z 419.675,A -85,B 0,C 180,E1 -31515.981,E2 -31515.981} C_VEL
LIN {X 0,Y 76.744,Z 421.16,A -85,B 0,C 180,E1 -31522.404,E2 -31522.404} C_VEL
LIN {X 0,Y 77.277,Z 424.061,A -85,B 0,C 180,E1 -31527.414,E2 -31527.414} C_VEL
LIN {X 0,Y 77.624,Z 425.919,A -85,B 0,C 180,E1 -31529.629,E2 -31529.629} C_VEL
LIN {X 0,Y 75.511,Z 438.414,A -85,B 0,C 180,E1 -31530.016,E2 -31530.016} C_VEL
LIN {X 0,Y 72.021,Z 451.223,A -85,B 0,C 180,E1 -31530.41,E2 -31530.41} C_VEL
LIN {X 0,Y 67.229,Z 463.595,A -85,B 0,C 180,E1 -31530.987,E2 -31530.987} C_VEL
LIN {X 0,Y 60.922,Z 475.907,A -85,B 0,C 180,E1 -31531.669,E2 -31531.669} C_VEL
LIN {X 0,Y 53.316,Z 487.481,A -85,B 0,C 180,E1 -31532.741,E2 -31532.741} C_VEL
LIN {X 0,Y 44.756,Z 497.982,A -85,B 0,C 180,E1 -31534.427,E2 -31534.427} C_VEL
LIN {X 0,Y 34.809,Z 507.847,A -85,B 0,C 180,E1 -31537.28,E2 -31537.28} C_VEL
LIN {X 0,Y 23.911,Z 516.554,A -85,B 0,C 180,E1 -31542.634,E2 -31542.634} C_VEL
LIN {X 0,Y 12.846,Z 523.829,A -85,B 0,C 180,E1 -31556.712,E2 -31556.712} C_VEL
LIN {X 0,Y 11,Z 524.92,A -85,B 0,C 180,E1 -31561.687,E2 -31561.687} C_VEL
LIN {X 0,Y 10.108,Z 525.112,A -85,B 0,C 180,E1 -31558.902,E2 -31558.902} C_VEL
LIN {X 0,Y 9.806,Z 524.581,A -85,B 0,C 180,E1 -31544.678,E2 -31544.678} C_VEL
LIN {X 0,Y 12.225,Z 522.812,A -85,B 0,C 180,E1 -31524.867,E2 -31524.867} C_VEL
LIN {X 0,Y 18.011,Z 519.283,A -85,B 0,C 180,E1 -31513.713,E2 -31513.713} C_VEL
LIN {X 0,Y 22.752,Z 516.2,A -85,B 0,C 180,E1 -31509.973,E2 -31509.973} C_VEL
LIN {X 0,Y 29.731,Z 511.085,A -85,B 0,C 180,E1 -31507.917,E2 -31507.917} C_VEL
LIN {X 0,Y 31.977,Z 509.207,A -85,B 0,C 180,E1 -31507.842,E2 -31507.842} C_VEL
LIN {X 0,Y 40.809,Z 501,A -85,B 0,C 180,E1 -31507.803,E2 -31507.803} C_VEL
LIN {X 0,Y 49.679,Z 490.922,A -85,B 0,C 180,E1 -31507.829,E2 -31507.829} C_VEL
LIN {X 0,Y 57.651,Z 479.58,A -85,B 0,C 180,E1 -31507.77,E2 -31507.77} C_VEL
LIN {X 0,Y 63.85,Z 468.525,A -85,B 0,C 180,E1 -31507.723,E2 -31507.723} C_VEL
LIN {X 0,Y 69.161,Z 456.276,A -85,B 0,C 180,E1 -31507.676,E2 -31507.676} C_VEL
LIN {X 0,Y 73.443,Z 442.409,A -85,B 0,C 180,E1 -31507.647,E2 -31507.647} C_VEL
LIN {X 0,Y 75.884,Z 429.913,A -85,B 0,C 180,E1 -31507.824,E2 -31507.824} C_VEL
LIN {X 0,Y 75.701,Z 427.061,A -85,B 0,C 180,E1 -31512.108,E2 -31512.108} C_VEL
LIN {X 0,Y 75.609,Z 426.674,A -85,B 0,C 180,E1 -31514.606,E2 -31514.606} C_VEL
LIN {X 0,Y 75.614,Z 427.753,A -85,B 0,C 180,E1 -31520.608,E2 -31520.608} C_VEL
LIN {X 0,Y 75.798,Z 429.907,A -85,B 0,C 180,E1 -31524.489,E2 -31524.489} C_VEL
LIN {X 0,Y 73.153,Z 442.928,A -85,B 0,C 180,E1 -31524.683,E2 -31524.683} C_VEL
LIN {X 0,Y 69.106,Z 455.922,A -85,B 0,C 180,E1 -31524.882,E2 -31524.882} C_VEL
LIN {X 0,Y 64.052,Z 467.639,A -85,B 0,C 180,E1 -31524.983,E2 -31524.983} C_VEL
LIN {X 0,Y 57.234,Z 479.8,A -85,B 0,C 180,E1 -31525.05,E2 -31525.05} C_VEL
LIN {X 0,Y 49.473,Z 490.811,A -85,B 0,C 180,E1 -31525.225,E2 -31525.225} C_VEL
LIN {X 0,Y 40.87,Z 500.615,A -85,B 0,C 180,E1 -31525.407,E2 -31525.407} C_VEL
LIN {X 0,Y 31.183,Z 509.626,A -85,B 0,C 180,E1 -31525.555,E2 -31525.555} C_VEL
LIN {X 0,Y 21.416,Z 517.051,A -85,B 0,C 180,E1 -31525.386,E2 -31525.386} C_VEL
LIN {X 0,Y 11.526,Z 523.183,A -85,B 0,C 180,E1 -31523.573,E2 -31523.573} C_VEL
LIN {X 0,Y 7.499,Z 525.327,A -85,B 0,C 180,E1 -31519.929,E2 -31519.929} C_VEL
LIN {X 0,Y 7.176,Z 525.543,A -85,B 0,C 180,E1 -31510.729,E2 -31510.729} C_VEL
LIN {X 0,Y 17.784,Z 519.573,A -85,B 0,C 180,E1 -31508.441,E2 -31508.441} C_VEL
LIN {X 0,Y 28.403,Z 512.124,A -85,B 0,C 180,E1 -31507.905,E2 -31507.905} C_VEL
LIN {X 0,Y 31.977,Z 509.207,A -85,B 0,C 180,E1 -31507.842,E2 -31507.842} C_VEL
LIN {X 0,Y 36.769,Z 504.857,A -85,B 0,C 180,E1 -31508.922,E2 -31508.922} C_VEL
LIN {X 0,Y 44.02,Z 497.07,A -85,B 0,C 180,E1 -31512.432,E2 -31512.432} C_VEL
LIN {X 0,Y 49.423,Z 490.443,A -85,B 0,C 180,E1 -31514.681,E2 -31514.681} C_VEL
LIN {X 0,Y 53.285,Z 485.143,A -85,B 0,C 180,E1 -31515.272,E2 -31515.272} C_VEL
LIN {X 0,Y 54.534,Z 483.317,A -85,B 0,C 180,E1 -31515.183,E2 -31515.183} C_VEL
LIN {X 0,Y 61.65,Z 471.452,A -85,B 0,C 180,E1 -31514.238,E2 -31514.238} C_VEL
LIN {X 0,Y 67.32,Z 459.15,A -85,B 0,C 180,E1 -31513.642,E2 -31513.642} C_VEL
LIN {X 0,Y 71.809,Z 445.977,A -85,B 0,C 180,E1 -31513.277,E2 -31513.277} C_VEL
LIN {X 0,Y 74.523,Z 434.08,A -85,B 0,C 180,E1 -31513.21,E2 -31513.21} C_VEL
LIN {X 0,Y 74.535,Z 433.795,A -85,B 0,C 180,E1 -31513.828,E2 -31513.828} C_VEL
LIN {X 0,Y 74.448,Z 434.172,A -85,B 0,C 180,E1 -31517.802,E2 -31517.802} C_VEL
LIN {X 0,Y 74.424,Z 434.591,A -85,B 0,C 180,E1 -31519.168,E2 -31519.168} C_VEL
LIN {X 0,Y 71.143,Z 448.059,A -85,B 0,C 180,E1 -31519.1,E2 -31519.1} C_VEL
LIN {X 0,Y 66.872,Z 460.153,A -85,B 0,C 180,E1 -31518.891,E2 -31518.891} C_VEL
LIN {X 0,Y 61.112,Z 472.397,A -85,B 0,C 180,E1 -31518.365,E2 -31518.365} C_VEL
LIN {X 0,Y 54.051,Z 483.986,A -85,B 0,C 180,E1 -31517.641,E2 -31517.641} C_VEL
LIN {X 0,Y 48.408,Z 491.673,A -85,B 0,C 180,E1 -31516.88,E2 -31516.88} C_VEL
LIN {X 0,Y 48.898,Z 491.08,A -85,B 0,C 180,E1 -31516.09,E2 -31516.09} C_VEL
LIN {X 0,Y 54.534,Z 483.317,A -85,B 0,C 180,E1 -31515.183,E2 -31515.183} C_VEL
LIN {X 0,Y 58.15,Z 484.455,A -85,B 0,C 180,E1 -31514.725,E2 -31514.725} C_VEL
LIN {X 0,Y 58.15,Z 600,A -85,B 0,C 180,E1 -31514.725,E2 -31514.725} C_VEL
LIN {X 0,Y 58.15,Z 600,A -85,B 0,C 180,E1 -31514.725,E2 -31514.725}

QRS_NEXT_CUT()

QRS_NEXT()
QRS_HOME()

END
